// TwinCAT 3 PLC project lighting
// ProgramVersion: 3.1.4023.0
// libraries:
//   Tc2_Standard, * (Beckhoff Automation GmbH)
//   Tc2_System, * (Beckhoff Automation GmbH)
//   Tc2_Utilities, * (Beckhoff Automation GmbH)
//   Tc3_EventLogger, * (Beckhoff Automation GmbH)
//   Tc3_Module, * (Beckhoff Automation GmbH)
//   VisuDialogs, * (System)
//   Tc3_DALI,3.13.0.0,Beckhoff Automation GmbH
// project tree:
//   Bridge/ FB_DALIBridge.TcPOU, GVL_DALIBridge.TcGVL
//   Bridge/Types/ E_DALIBridgeCommand.TcTLEO, ST_DALIBridgeInputEvent.TcDUT, ST_DALIBridgeInputEventParams.TcDUT, ST_DALIBridgeNotification.TcDUT, ST_DALIBridgeRequest.TcDUT, ST_DALIBridgeResponse.TcDUT, U_ReinterpretDALIEnum.TcDUT
//   / BRIDGE_TASK.TcTTO, GlobalTextList.TcGTLO
//   GVLs/ GVL_Bridges.TcGVL, GVL_Variant.TcGVL
//   POUs/ MAIN.TcPOU
//   Tc3_DALI_PLC_Commissioning_Tool/ COMM_TASK.TcTTO, GlobalTextList_1.TcGTLO, ImagePool.TcIPO (not stored), VisualizationManager.TcVMO (not stored), VISU_TASK.TcTTO
//   Tc3_DALI_PLC_Commissioning_Tool/DUTs/ E_DALIExtendedFadeTime.TcTLEO, ST_DALI102Parameters.TcDUT, ST_DALI103Parameters.TcDUT, ST_DALIMemoryBank.TcDUT
//   Tc3_DALI_PLC_Commissioning_Tool/GVLs/ GVL.TcGVL, GVL_Internal.TcGVL
//   Tc3_DALI_PLC_Commissioning_Tool/POUs/ Communication.TcPOU, DALI_Commissioning.TcPOU, MAIN_Comissioning.TcPOU
//   Tc3_DALI_PLC_Commissioning_Tool/POUs/DALI_PLC_Commissioning/ FB_Part102Addressing.TcPOU, FB_Part102Commands.TcPOU (not stored), FB_Part102Groups.TcPOU, FB_Part102MemoryPages.TcPOU, FB_Part102Parameters.TcPOU, FB_Part102Scenes.TcPOU, FB_Part102SetFading.TcPOU, FB_Part103Addressing.TcPOU, FB_Part103MemoryPages.TcPOU, FB_Part103Parameters.TcPOU, FB_Part207ParametersLED.TcPOU, FB_Part207StatusLED.TcPOU, FB_Part300GenericDevice.TcPOU, FB_Part301PushButton.TcPOU, FB_Part302AbsoluteInputDevice.TcPOU, FB_Part303OccupancySensor.TcPOU, FB_Part304LightSensor.TcPOU
//   Tc3_DALI_PLC_Commissioning_Tool/Version/ Global_Version.TcGVL
//   Tc3_DALI_PLC_Commissioning_Tool/VISUs/TextLists/ CommandOnTerminalEvent.TcTLO, DimmingCurve.TcTLO, EventPriority.TcTLO, EventScheme.TcTLO, ExtendedFadeTime.TcTLO, FadeRate.TcTLO, FadeTime.TcTLO, FastFadeTime.TcTLO, TextList_Dialogs.TcTLO
//   Tc3_DALI_PLC_Commissioning_Tool/VISUs/ Visu_DALICommissioning.TcVIS
//   Tc3_DALI_PLC_Commissioning_Tool/VISUs/Visu_DALICommissioning/ Visu_KL6821Configuration.TcVIS, Visu_Part102Addressing.TcVIS, Visu_Part102Commands.TcVIS, Visu_Part102Groups.TcVIS, Visu_Part102MemoryBank.TcVIS, Visu_Part102Parameters.TcVIS, Visu_Part102Scenes.TcVIS, Visu_Part102SetFading.TcVIS, Visu_Part103Addressing.TcVIS, Visu_Part103MemoryBank.TcVIS, Visu_Part103Parameters.TcVIS, Visu_Part207Parameters.TcVIS, Visu_Part207Status.TcVIS, Visu_Part300GenericDevice.TcVIS, Visu_Part301PushButton.TcVIS, Visu_Part302AbsoluteInputDevice.TcVIS, Visu_Part303OccupancySensor.TcVIS, Visu_Part304LightSensor.TcVIS
// real-time tasks:
//   TASK VISU_TASK: cycle T#80ms, priority 30, ADS port 353
//   TASK BRIDGE_TASK: cycle T#8ms, priority 3, ADS port 350
//   TASK COMM_TASK: cycle T#2ms, priority 2, ADS port 351
// I/O:
//   DEVICE Device 1 (EtherCAT), AmsNetId 5.109.178.35.2.1
//     Term 1 (EK1200) [EK1200-5000 EtherCAT Power supply (2A E-Bus)]
//       Junction 1 (EK1122) [EK1122 2 port EtherCAT junction] (disabled)
//         Tenant 1 Coupler (BK1150) (disabled)
//         Tenant 2 Coupler (BK1150)
//       Junction 2  (EK1122) [EK1122 2 port EtherCAT junction] (disabled)
//         Tenant 3 Coupler (BK1150)
//         Tenant 4 Coupler (BK1150)
//       Junction 3 (EK1122) [EK1122 2 port EtherCAT junction]
//         Life Safety Coupler (BK1150) (disabled)
//       Landlord Coupler (BK1250)
// variable links:
//   lighting Instance <-> Device 1 (EtherCAT)/Term 1 (EK1200)/Junction 1 (EK1122)/Tenant 1 Coupler (BK1150)
//     COMM_TASK Inputs/GVL.aKL6821InData[1] @bit 16 <-> T1 Bus 1 (KL6821)/Channel 1/Data In 0
//     COMM_TASK Inputs/GVL.aKL6821InData[1] @bit 24 <-> T1 Bus 1 (KL6821)/Channel 1/Data In 1
//     COMM_TASK Inputs/GVL.aKL6821InData[1] @bit 32 <-> T1 Bus 1 (KL6821)/Channel 1/Data In 2
//     COMM_TASK Inputs/GVL.aKL6821InData[1] @bit 40 <-> T1 Bus 1 (KL6821)/Channel 1/Data In 3
//     COMM_TASK Inputs/GVL.aKL6821InData[2] @bit 16 <-> T1 Bus 2 (KL6821)/Channel 1/Data In 0
//     COMM_TASK Inputs/GVL.aKL6821InData[2] @bit 24 <-> T1 Bus 2 (KL6821)/Channel 1/Data In 1
//     COMM_TASK Inputs/GVL.aKL6821InData[2] @bit 32 <-> T1 Bus 2 (KL6821)/Channel 1/Data In 2
//     COMM_TASK Inputs/GVL.aKL6821InData[2] @bit 40 <-> T1 Bus 2 (KL6821)/Channel 1/Data In 3
//     COMM_TASK Inputs/GVL.aKL6821InData[1] <-> T1 Bus 1 (KL6821)/Channel 1/State
//     COMM_TASK Inputs/GVL.aKL6821InData[2] <-> T1 Bus 2 (KL6821)/Channel 1/State
//     COMM_TASK Outputs/GVL.aKL6821OutData[1] <-> T1 Bus 1 (KL6821)/Channel 1/Ctrl
//     COMM_TASK Outputs/GVL.aKL6821OutData[2] <-> T1 Bus 2 (KL6821)/Channel 1/Ctrl
//     COMM_TASK Outputs/GVL.aKL6821OutData[1] @bit 16 <-> T1 Bus 1 (KL6821)/Channel 1/Data Out 0
//     COMM_TASK Outputs/GVL.aKL6821OutData[1] @bit 24 <-> T1 Bus 1 (KL6821)/Channel 1/Data Out 1
//     COMM_TASK Outputs/GVL.aKL6821OutData[1] @bit 32 <-> T1 Bus 1 (KL6821)/Channel 1/Data Out 2
//     COMM_TASK Outputs/GVL.aKL6821OutData[1] @bit 40 <-> T1 Bus 1 (KL6821)/Channel 1/Data Out 3
//     COMM_TASK Outputs/GVL.aKL6821OutData[2] @bit 16 <-> T1 Bus 2 (KL6821)/Channel 1/Data Out 0
//     COMM_TASK Outputs/GVL.aKL6821OutData[2] @bit 24 <-> T1 Bus 2 (KL6821)/Channel 1/Data Out 1
//     COMM_TASK Outputs/GVL.aKL6821OutData[2] @bit 32 <-> T1 Bus 2 (KL6821)/Channel 1/Data Out 2
//     COMM_TASK Outputs/GVL.aKL6821OutData[2] @bit 40 <-> T1 Bus 2 (KL6821)/Channel 1/Data Out 3
//   lighting Instance <-> Device 1 (EtherCAT)/Term 1 (EK1200)/Junction 1 (EK1122)/Tenant 2 Coupler (BK1150)
//     COMM_TASK Inputs/GVL.aKL6821InData[3] @bit 16 <-> T2 Bus 1 (KL6821)/Channel 1/Data In 0
//     COMM_TASK Inputs/GVL.aKL6821InData[3] @bit 24 <-> T2 Bus 1 (KL6821)/Channel 1/Data In 1
//     COMM_TASK Inputs/GVL.aKL6821InData[3] @bit 32 <-> T2 Bus 1 (KL6821)/Channel 1/Data In 2
//     COMM_TASK Inputs/GVL.aKL6821InData[3] @bit 40 <-> T2 Bus 1 (KL6821)/Channel 1/Data In 3
//     COMM_TASK Inputs/GVL.aKL6821InData[5] @bit 16 <-> T2 Bus 3 (KL6821)/Channel 1/Data In 0
//     COMM_TASK Inputs/GVL.aKL6821InData[5] @bit 24 <-> T2 Bus 3 (KL6821)/Channel 1/Data In 1
//     COMM_TASK Inputs/GVL.aKL6821InData[5] @bit 32 <-> T2 Bus 3 (KL6821)/Channel 1/Data In 2
//     COMM_TASK Inputs/GVL.aKL6821InData[5] @bit 40 <-> T2 Bus 3 (KL6821)/Channel 1/Data In 3
//     COMM_TASK Inputs/GVL.aKL6821InData[3] <-> T2 Bus 1 (KL6821)/Channel 1/State
//     COMM_TASK Inputs/GVL.aKL6821InData[5] <-> T2 Bus 3 (KL6821)/Channel 1/State
//     COMM_TASK Inputs/GVL.aKL6821InData[4]/aData[{0..3}] <-> T2 Bus 2 (KL6821)/Channel 1/Data In {0..3}  (4 links)
//     COMM_TASK Inputs/GVL.aKL6821InData[4]/nStatus <-> T2 Bus 2 (KL6821)/Channel 1/State
//     COMM_TASK Outputs/GVL.aKL6821OutData[3] <-> T2 Bus 1 (KL6821)/Channel 1/Ctrl
//     COMM_TASK Outputs/GVL.aKL6821OutData[4] <-> T2 Bus 2 (KL6821)/Channel 1/Ctrl
//     COMM_TASK Outputs/GVL.aKL6821OutData[5] <-> T2 Bus 3 (KL6821)/Channel 1/Ctrl
//     COMM_TASK Outputs/GVL.aKL6821OutData[3] @bit 16 <-> T2 Bus 1 (KL6821)/Channel 1/Data Out 0
//     COMM_TASK Outputs/GVL.aKL6821OutData[3] @bit 24 <-> T2 Bus 1 (KL6821)/Channel 1/Data Out 1
//     COMM_TASK Outputs/GVL.aKL6821OutData[3] @bit 32 <-> T2 Bus 1 (KL6821)/Channel 1/Data Out 2
//     COMM_TASK Outputs/GVL.aKL6821OutData[3] @bit 40 <-> T2 Bus 1 (KL6821)/Channel 1/Data Out 3
//     COMM_TASK Outputs/GVL.aKL6821OutData[4] @bit 16 <-> T2 Bus 2 (KL6821)/Channel 1/Data Out 0
//     COMM_TASK Outputs/GVL.aKL6821OutData[4] @bit 24 <-> T2 Bus 2 (KL6821)/Channel 1/Data Out 1
//     COMM_TASK Outputs/GVL.aKL6821OutData[4] @bit 32 <-> T2 Bus 2 (KL6821)/Channel 1/Data Out 2
//     COMM_TASK Outputs/GVL.aKL6821OutData[4] @bit 40 <-> T2 Bus 2 (KL6821)/Channel 1/Data Out 3
//     COMM_TASK Outputs/GVL.aKL6821OutData[5] @bit 16 <-> T2 Bus 3 (KL6821)/Channel 1/Data Out 0
//     COMM_TASK Outputs/GVL.aKL6821OutData[5] @bit 24 <-> T2 Bus 3 (KL6821)/Channel 1/Data Out 1
//     COMM_TASK Outputs/GVL.aKL6821OutData[5] @bit 32 <-> T2 Bus 3 (KL6821)/Channel 1/Data Out 2
//     COMM_TASK Outputs/GVL.aKL6821OutData[5] @bit 40 <-> T2 Bus 3 (KL6821)/Channel 1/Data Out 3
//   lighting Instance <-> Device 1 (EtherCAT)/Term 1 (EK1200)/Junction 2  (EK1122)/Tenant 3 Coupler (BK1150)
//     COMM_TASK Inputs/GVL.aKL6821InData[6] @bit 16 <-> T3 Bus 1 (KL6821)/Channel 1/Data In 0
//     COMM_TASK Inputs/GVL.aKL6821InData[6] @bit 24 <-> T3 Bus 1 (KL6821)/Channel 1/Data In 1
//     COMM_TASK Inputs/GVL.aKL6821InData[6] @bit 32 <-> T3 Bus 1 (KL6821)/Channel 1/Data In 2
//     COMM_TASK Inputs/GVL.aKL6821InData[6] @bit 40 <-> T3 Bus 1 (KL6821)/Channel 1/Data In 3
//     COMM_TASK Inputs/GVL.aKL6821InData[7] @bit 16 <-> T3 Bus 2 (KL6821)/Channel 1/Data In 0
//     COMM_TASK Inputs/GVL.aKL6821InData[7] @bit 24 <-> T3 Bus 2 (KL6821)/Channel 1/Data In 1
//     COMM_TASK Inputs/GVL.aKL6821InData[7] @bit 32 <-> T3 Bus 2 (KL6821)/Channel 1/Data In 2
//     COMM_TASK Inputs/GVL.aKL6821InData[7] @bit 40 <-> T3 Bus 2 (KL6821)/Channel 1/Data In 3
//     COMM_TASK Inputs/GVL.aKL6821InData[6] <-> T3 Bus 1 (KL6821)/Channel 1/State
//     COMM_TASK Inputs/GVL.aKL6821InData[7] <-> T3 Bus 2 (KL6821)/Channel 1/State
//     COMM_TASK Outputs/GVL.aKL6821OutData[6] <-> T3 Bus 1 (KL6821)/Channel 1/Ctrl
//     COMM_TASK Outputs/GVL.aKL6821OutData[7] <-> T3 Bus 2 (KL6821)/Channel 1/Ctrl
//     COMM_TASK Outputs/GVL.aKL6821OutData[6] @bit 16 <-> T3 Bus 1 (KL6821)/Channel 1/Data Out 0
//     COMM_TASK Outputs/GVL.aKL6821OutData[6] @bit 24 <-> T3 Bus 1 (KL6821)/Channel 1/Data Out 1
//     COMM_TASK Outputs/GVL.aKL6821OutData[6] @bit 32 <-> T3 Bus 1 (KL6821)/Channel 1/Data Out 2
//     COMM_TASK Outputs/GVL.aKL6821OutData[6] @bit 40 <-> T3 Bus 1 (KL6821)/Channel 1/Data Out 3
//     COMM_TASK Outputs/GVL.aKL6821OutData[7] @bit 16 <-> T3 Bus 2 (KL6821)/Channel 1/Data Out 0
//     COMM_TASK Outputs/GVL.aKL6821OutData[7] @bit 24 <-> T3 Bus 2 (KL6821)/Channel 1/Data Out 1
//     COMM_TASK Outputs/GVL.aKL6821OutData[7] @bit 32 <-> T3 Bus 2 (KL6821)/Channel 1/Data Out 2
//     COMM_TASK Outputs/GVL.aKL6821OutData[7] @bit 40 <-> T3 Bus 2 (KL6821)/Channel 1/Data Out 3
//   lighting Instance <-> Device 1 (EtherCAT)/Term 1 (EK1200)/Junction 2  (EK1122)/Tenant 4 Coupler (BK1150)
//     COMM_TASK Inputs/GVL.aKL6821InData[8] @bit 16 <-> T4 Bus 1 (KL6821)/Channel 1/Data In 0
//     COMM_TASK Inputs/GVL.aKL6821InData[8] @bit 24 <-> T4 Bus 1 (KL6821)/Channel 1/Data In 1
//     COMM_TASK Inputs/GVL.aKL6821InData[8] @bit 32 <-> T4 Bus 1 (KL6821)/Channel 1/Data In 2
//     COMM_TASK Inputs/GVL.aKL6821InData[8] @bit 40 <-> T4 Bus 1 (KL6821)/Channel 1/Data In 3
//     COMM_TASK Inputs/GVL.aKL6821InData[9] @bit 16 <-> T4 Bus 2 (KL6821)/Channel 1/Data In 0
//     COMM_TASK Inputs/GVL.aKL6821InData[9] @bit 24 <-> T4 Bus 2 (KL6821)/Channel 1/Data In 1
//     COMM_TASK Inputs/GVL.aKL6821InData[9] @bit 32 <-> T4 Bus 2 (KL6821)/Channel 1/Data In 2
//     COMM_TASK Inputs/GVL.aKL6821InData[9] @bit 40 <-> T4 Bus 2 (KL6821)/Channel 1/Data In 3
//     COMM_TASK Inputs/GVL.aKL6821InData[8] <-> T4 Bus 1 (KL6821)/Channel 1/State
//     COMM_TASK Inputs/GVL.aKL6821InData[9] <-> T4 Bus 2 (KL6821)/Channel 1/State
//     COMM_TASK Outputs/GVL.aKL6821OutData[8] <-> T4 Bus 1 (KL6821)/Channel 1/Ctrl
//     COMM_TASK Outputs/GVL.aKL6821OutData[9] <-> T4 Bus 2 (KL6821)/Channel 1/Ctrl
//     COMM_TASK Outputs/GVL.aKL6821OutData[8] @bit 16 <-> T4 Bus 1 (KL6821)/Channel 1/Data Out 0
//     COMM_TASK Outputs/GVL.aKL6821OutData[8] @bit 24 <-> T4 Bus 1 (KL6821)/Channel 1/Data Out 1
//     COMM_TASK Outputs/GVL.aKL6821OutData[8] @bit 32 <-> T4 Bus 1 (KL6821)/Channel 1/Data Out 2
//     COMM_TASK Outputs/GVL.aKL6821OutData[8] @bit 40 <-> T4 Bus 1 (KL6821)/Channel 1/Data Out 3
//     COMM_TASK Outputs/GVL.aKL6821OutData[9] @bit 16 <-> T4 Bus 2 (KL6821)/Channel 1/Data Out 0
//     COMM_TASK Outputs/GVL.aKL6821OutData[9] @bit 24 <-> T4 Bus 2 (KL6821)/Channel 1/Data Out 1
//     COMM_TASK Outputs/GVL.aKL6821OutData[9] @bit 32 <-> T4 Bus 2 (KL6821)/Channel 1/Data Out 2
//     COMM_TASK Outputs/GVL.aKL6821OutData[9] @bit 40 <-> T4 Bus 2 (KL6821)/Channel 1/Data Out 3
//   lighting Instance <-> Device 1 (EtherCAT)/Term 1 (EK1200)/Junction 3 (EK1122)/Life Safety Coupler (BK1150)
//     COMM_TASK Inputs/GVL.aKL6821InData[10] @bit {16..40 step 8} <-> LS Bus (KL6821)/Channel 1/Data In {0..3}  (4 links)
//     COMM_TASK Inputs/GVL.aKL6821InData[10] <-> LS Bus (KL6821)/Channel 1/State
//     COMM_TASK Outputs/GVL.aKL6821OutData[10] <-> LS Bus (KL6821)/Channel 1/Ctrl
//     COMM_TASK Outputs/GVL.aKL6821OutData[10] @bit {16..40 step 8} <-> LS Bus (KL6821)/Channel 1/Data Out {0..3}  (4 links)
//   lighting Instance <-> Device 1 (EtherCAT)/Term 1 (EK1200)/Landlord Coupler (BK1250)
//     COMM_TASK Inputs/GVL.aKL6821InData[11] @bit 16 <-> LL Bus 1 (KL6821)/Channel 1/Data In 0
//     COMM_TASK Inputs/GVL.aKL6821InData[11] @bit 24 <-> LL Bus 1 (KL6821)/Channel 1/Data In 1
//     COMM_TASK Inputs/GVL.aKL6821InData[11] @bit 32 <-> LL Bus 1 (KL6821)/Channel 1/Data In 2
//     COMM_TASK Inputs/GVL.aKL6821InData[11] @bit 40 <-> LL Bus 1 (KL6821)/Channel 1/Data In 3
//     COMM_TASK Inputs/GVL.aKL6821InData[12] @bit 16 <-> LL Bus 2 (KL6821)/Channel 1/Data In 0
//     COMM_TASK Inputs/GVL.aKL6821InData[12] @bit 24 <-> LL Bus 2 (KL6821)/Channel 1/Data In 1
//     COMM_TASK Inputs/GVL.aKL6821InData[12] @bit 32 <-> LL Bus 2 (KL6821)/Channel 1/Data In 2
//     COMM_TASK Inputs/GVL.aKL6821InData[12] @bit 40 <-> LL Bus 2 (KL6821)/Channel 1/Data In 3
//     COMM_TASK Inputs/GVL.aKL6821InData[13] @bit 16 <-> LL Bus 3 (KL6821)/Channel 1/Data In 0
//     COMM_TASK Inputs/GVL.aKL6821InData[13] @bit 24 <-> LL Bus 3 (KL6821)/Channel 1/Data In 1
//     COMM_TASK Inputs/GVL.aKL6821InData[13] @bit 32 <-> LL Bus 3 (KL6821)/Channel 1/Data In 2
//     COMM_TASK Inputs/GVL.aKL6821InData[13] @bit 40 <-> LL Bus 3 (KL6821)/Channel 1/Data In 3
//     COMM_TASK Inputs/GVL.aKL6821InData[14] @bit 16 <-> LL Bus 4 (KL6821)/Channel 1/Data In 0
//     COMM_TASK Inputs/GVL.aKL6821InData[14] @bit 24 <-> LL Bus 4 (KL6821)/Channel 1/Data In 1
//     COMM_TASK Inputs/GVL.aKL6821InData[14] @bit 32 <-> LL Bus 4 (KL6821)/Channel 1/Data In 2
//     COMM_TASK Inputs/GVL.aKL6821InData[14] @bit 40 <-> LL Bus 4 (KL6821)/Channel 1/Data In 3
//     COMM_TASK Inputs/GVL.aKL6821InData[15] @bit 16 <-> LL Bus 5 (KL6821)/Channel 1/Data In 0
//     COMM_TASK Inputs/GVL.aKL6821InData[15] @bit 24 <-> LL Bus 5 (KL6821)/Channel 1/Data In 1
//     COMM_TASK Inputs/GVL.aKL6821InData[15] @bit 32 <-> LL Bus 5 (KL6821)/Channel 1/Data In 2
//     COMM_TASK Inputs/GVL.aKL6821InData[15] @bit 40 <-> LL Bus 5 (KL6821)/Channel 1/Data In 3
//     COMM_TASK Inputs/GVL.aKL6821InData[16] @bit 16 <-> LL Bus 6 (KL6821)/Channel 1/Data In 0
//     COMM_TASK Inputs/GVL.aKL6821InData[16] @bit 24 <-> LL Bus 6 (KL6821)/Channel 1/Data In 1
//     COMM_TASK Inputs/GVL.aKL6821InData[16] @bit 32 <-> LL Bus 6 (KL6821)/Channel 1/Data In 2
//     COMM_TASK Inputs/GVL.aKL6821InData[16] @bit 40 <-> LL Bus 6 (KL6821)/Channel 1/Data In 3
//     COMM_TASK Inputs/GVL.aKL6821InData[{11..16}] <-> LL Bus {1..6} (KL6821)/Channel 1/State  (6 links)
//     COMM_TASK Outputs/GVL.aKL6821OutData[{11..16}] <-> LL Bus {1..6} (KL6821)/Channel 1/Ctrl  (6 links)
//     COMM_TASK Outputs/GVL.aKL6821OutData[11] @bit 16 <-> LL Bus 1 (KL6821)/Channel 1/Data Out 0
//     COMM_TASK Outputs/GVL.aKL6821OutData[11] @bit 24 <-> LL Bus 1 (KL6821)/Channel 1/Data Out 1
//     COMM_TASK Outputs/GVL.aKL6821OutData[11] @bit 32 <-> LL Bus 1 (KL6821)/Channel 1/Data Out 2
//     COMM_TASK Outputs/GVL.aKL6821OutData[11] @bit 40 <-> LL Bus 1 (KL6821)/Channel 1/Data Out 3
//     COMM_TASK Outputs/GVL.aKL6821OutData[12] @bit 16 <-> LL Bus 2 (KL6821)/Channel 1/Data Out 0
//     COMM_TASK Outputs/GVL.aKL6821OutData[12] @bit 24 <-> LL Bus 2 (KL6821)/Channel 1/Data Out 1
//     COMM_TASK Outputs/GVL.aKL6821OutData[12] @bit 32 <-> LL Bus 2 (KL6821)/Channel 1/Data Out 2
//     COMM_TASK Outputs/GVL.aKL6821OutData[12] @bit 40 <-> LL Bus 2 (KL6821)/Channel 1/Data Out 3
//     COMM_TASK Outputs/GVL.aKL6821OutData[13] @bit 16 <-> LL Bus 3 (KL6821)/Channel 1/Data Out 0
//     COMM_TASK Outputs/GVL.aKL6821OutData[13] @bit 24 <-> LL Bus 3 (KL6821)/Channel 1/Data Out 1
//     COMM_TASK Outputs/GVL.aKL6821OutData[13] @bit 32 <-> LL Bus 3 (KL6821)/Channel 1/Data Out 2
//     COMM_TASK Outputs/GVL.aKL6821OutData[13] @bit 40 <-> LL Bus 3 (KL6821)/Channel 1/Data Out 3
//     COMM_TASK Outputs/GVL.aKL6821OutData[14] @bit 16 <-> LL Bus 4 (KL6821)/Channel 1/Data Out 0
//     COMM_TASK Outputs/GVL.aKL6821OutData[14] @bit 24 <-> LL Bus 4 (KL6821)/Channel 1/Data Out 1
//     COMM_TASK Outputs/GVL.aKL6821OutData[14] @bit 32 <-> LL Bus 4 (KL6821)/Channel 1/Data Out 2
//     COMM_TASK Outputs/GVL.aKL6821OutData[14] @bit 40 <-> LL Bus 4 (KL6821)/Channel 1/Data Out 3
//     COMM_TASK Outputs/GVL.aKL6821OutData[15] @bit 16 <-> LL Bus 5 (KL6821)/Channel 1/Data Out 0
//     COMM_TASK Outputs/GVL.aKL6821OutData[15] @bit 24 <-> LL Bus 5 (KL6821)/Channel 1/Data Out 1
//     COMM_TASK Outputs/GVL.aKL6821OutData[15] @bit 32 <-> LL Bus 5 (KL6821)/Channel 1/Data Out 2
//     COMM_TASK Outputs/GVL.aKL6821OutData[15] @bit 40 <-> LL Bus 5 (KL6821)/Channel 1/Data Out 3
//     COMM_TASK Outputs/GVL.aKL6821OutData[16] @bit 16 <-> LL Bus 6 (KL6821)/Channel 1/Data Out 0
//     COMM_TASK Outputs/GVL.aKL6821OutData[16] @bit 24 <-> LL Bus 6 (KL6821)/Channel 1/Data Out 1
//     COMM_TASK Outputs/GVL.aKL6821OutData[16] @bit 32 <-> LL Bus 6 (KL6821)/Channel 1/Data Out 2
//     COMM_TASK Outputs/GVL.aKL6821OutData[16] @bit 40 <-> LL Bus 6 (KL6821)/Channel 1/Data Out 3

CONFIGURATION lighting
    RESOURCE PLC ON TwinCAT3
        TASK BRIDGE_TASK(INTERVAL := T#8ms, PRIORITY := 3);
        TASK COMM_TASK(INTERVAL := T#2ms, PRIORITY := 2);
        TASK VISU_TASK(INTERVAL := T#80ms, PRIORITY := 30);
        PROGRAM MAIN WITH BRIDGE_TASK : MAIN;
        PROGRAM MAIN_Comissioning WITH BRIDGE_TASK : MAIN_Comissioning;
        PROGRAM Communication WITH COMM_TASK : Communication;
        PROGRAM VisuElems_Visu_Prg WITH VISU_TASK : VisuElems.Visu_Prg;
    END_RESOURCE
END_CONFIGURATION

// ---- Bridge/Types/E_DALIBridgeCommand.TcTLEO
{attribute 'qualified_only'}
{attribute 'strict'}
TYPE E_DALIBridgeCommand :
(
	idle						:= 0,
	directArcPowerControl		:= 1,
	queryActualLevel			:= 2,
	queryStatus					:= 3,
	setEventScheme				:= 4,
	queryEventScheme			:= 5,
	setEventFilter				:= 6,
	queryEventFilter			:= 7,
	identifyDevice102			:= 8,
	identifyDevice103			:= 9,
	enableInstance				:= 10,
	goToScene					:= 11,
	setFadeTime					:= 12,
	queryInputValue				:= 13,
	queryBatteryCharge			:= 14,
	queryDurationTestResult		:= 15,
	queryEmergencyMode			:= 16,
	queryEmergencyStatus		:= 17,
	queryFailureStatus			:= 18,
	queryRatedDuration			:= 19,
	queryTestTiming				:= 20,
	resetDurationTestDoneFlag	:= 21,
	resetFunctionTestDoneFlag	:= 22,
	startDurationTest			:= 23,
	startFunctionTest			:= 24,
	stopTest					:= 25,
	setDurationTestInterval		:= 26,
	setFunctionTestInterval		:= 27,
	startIdentification202		:= 28,
	queryGroups					:= 29,
	addToGroup					:= 30,
	removeFromGroup				:= 31,
	enabledDeviceType			:= 32,
	
	testCommand := 100
);
END_TYPE

// ---- Bridge/Types/ST_DALIBridgeInputEvent.TcDUT
TYPE ST_DALIBridgeInputEvent :
STRUCT
	parameters : ST_DALIBridgeInputEventParams;
	error      : BOOL;
	status     : UDINT;
	message    : STRING(255);
	data       : WORD;
END_STRUCT
END_TYPE

// ---- Bridge/Types/ST_DALIBridgeInputEventParams.TcDUT
TYPE ST_DALIBridgeInputEventParams :
STRUCT
	eventScheme 	: E_DALIEventScheme;
	addressInfo1 	: BYTE;
	addressInfo2 	: BYTE;
END_STRUCT
END_TYPE

// ---- Bridge/Types/ST_DALIBridgeNotification.TcDUT
TYPE ST_DALIBridgeNotification :
STRUCT
	valid 				: BOOL;
	sequence 			: ULINT;
	nInputEvents		: BYTE;
	inputEvents 		: ARRAY [0..GVL_DALIBridge.maxInputEventsPerNotification-1] OF ST_DALIBridgeInputEvent;
END_STRUCT
END_TYPE

// ---- Bridge/Types/ST_DALIBridgeRequest.TcDUT
TYPE ST_DALIBridgeRequest :
STRUCT
	command 			: E_DALIBridgeCommand := E_DALIBridgeCommand.idle;
	address 			: BYTE;
	addressType 		: E_DALIAddressType;
	instanceAddress 	: BYTE;
	instanceAddressType : E_DALIInstanceAddressType;
	data            	: BYTE;
END_STRUCT
END_TYPE

// ---- Bridge/Types/ST_DALIBridgeResponse.TcDUT
TYPE ST_DALIBridgeResponse :
STRUCT
	valid       : BOOL := FALSE; 	// True if the struct contains valid data.
	sequence 	: ULINT;			// Same as the sequence number returned when calling RpcRequest
	error       : BOOL;				// True if an error condition ocurred. If error is false but status is nonzero, a warning occurred.
	status      : UDINT;			// Status code returned by the operation
	message     : STRING(255);		// Human-readable error message
	data 		: LWORD;			// Data returned by a DALI read command. If the command does not read data, then ignore this field.
END_STRUCT
END_TYPE

// ---- Bridge/Types/U_ReinterpretDALIEnum.TcDUT
TYPE U_ReinterpretDALIEnum :
UNION
	raw				: BYTE;
	eventScheme 	: E_DALIEventScheme;
	fadeTime		: E_DALIFadeTime;
	testTiming      : E_DALITestTiming;
	deviceType		: E_DALIDeviceType;
END_UNION
END_TYPE

// ---- Tc3_DALI_PLC_Commissioning_Tool/DUTs/E_DALIExtendedFadeTime.TcTLEO
{attribute 'qualified_only'}
{attribute 'strict'}
TYPE E_DALIExtendedFadeTime :
(
	NoFade := 0,
	onehundred := 1,
	twohundred := 2,
	threehundred := 3,
	fourhundred := 4,
	fivehundred := 5,
	sixhundred := 6,
	sevenhundred := 7,
	eighthundred := 8,
	ninehundred := 9,
	onethousand := 10,
	onethousandonehundred := 11,
	onethousandtwohundred := 12,
	onethousandthreehundred := 13,
	onethousandfourhundred := 14,
	onethousandfivehundred := 15,
	onethousandsixhundred	:= 16,
	onesecond := 17,
	twoseconds := 18,
	threeseconds := 19,
	fourseconds := 20,
	fiveseconds := 21,
	sixseconds := 22,
	sevenseconds := 23,
	eightseconds := 24,
	nineseconds := 25,
	tenseconds := 26,
	elevenseconds := 27,
	twelveseconds := 28,
	thirteenseconds := 29,
	fourteenseconds := 30,
	fifteenseconds := 31,
	sixteenseconds := 32,
	ten1seconds := 33,
	twentyseconds := 34,
	thirtyseconds := 35,
	fourtyseconds := 36,
	fiftyseconds := 37,
	sixtyseconds := 38,
	seventyseconds := 39,
	eightyseconds := 40,
	ninetyseconds := 41,
	onehundredseconds := 42,
	onehundredtenseconds := 43,
	onehundredtwentyseconds := 44,
	onehundredthirtyseconds := 45,
	onehundredfourtyseconds := 46,
	onehundredfiftyseconds := 47,
	onehundredsixtyseconds := 48,
	oneminute := 49,
	twominutes := 50,
	threeminutes := 51,
	fourminutes := 52,
	fiveminutes := 53,
	sixminutes := 54,
	sevenminutes := 55,
	eightminutes := 56,
	nineminutes := 57,
	tenminutes := 58,
	elevenminutes := 59,
	twelveminutes := 60,
	thirteenminutes := 61,
	fourteenminutes := 62,
	fifteenminutes := 63,
	sixteenminutes := 64,
	unknown := 255
);
END_TYPE

// ---- Tc3_DALI_PLC_Commissioning_Tool/DUTs/ST_DALI102Parameters.TcDUT
TYPE ST_DALI102Parameters :
STRUCT
	nShortAddress			:	BYTE; // 255: no short address
	nActualLevel			:	BYTE;
	nMinLevel				:	BYTE;
	nMaxLevel				: 	BYTE;
	eFadeRate				:	E_DALIFadeRate;
	eFadeTime				:	E_DALIFadeTime;
	nPowerOnLevel			:	BYTE;
	nSystemFailureLevel		:	BYTE;
	nPhysicalMinimum		:	BYTE;
	sDeviceTypes			:	STRING[100];
END_STRUCT
END_TYPE

// ---- Tc3_DALI_PLC_Commissioning_Tool/DUTs/ST_DALI103Parameters.TcDUT
TYPE ST_DALI103Parameters :
STRUCT
	nOperatingMode			:	BYTE;
	sInstanceType0			:	STRING;
	sInstanceType1			:	STRING;
	sInstanceType2			:	STRING;
	sInstanceType3			:	STRING;
	sInstanceType4			:	STRING;
END_STRUCT
END_TYPE

// ---- Tc3_DALI_PLC_Commissioning_Tool/DUTs/ST_DALIMemoryBank.TcDUT
TYPE ST_DALIMemoryBank :
STRUCT
	sOffset			:	STRING(20);
	sName			:	STRING(255);
	nValueDec		:	BYTE;
	nValueHex		:	STRING(20);
END_STRUCT
END_TYPE

// ---- Bridge/GVL_DALIBridge.TcGVL
{attribute 'qualified_only'}
VAR_GLOBAL

END_VAR
VAR_GLOBAL CONSTANT
	maxInputEventListeners: INT := 64;
	maxInputEventsPerNotification: INT := 4;
END_VAR

// ---- GVLs/GVL_Bridges.TcGVL
{attribute 'qualified_only'}
VAR_GLOBAL
	// Landlord Buses
	bus_LL1_bridge			: FB_DALIBridge(Communication.aKL6821Communication[11]);
	bus_LL1_response		: ST_DALIBridgeResponse;
	bus_LL1_notification	: ST_DALIBridgeNotification;
	
	bus_LL2_bridge			: FB_DALIBridge(Communication.aKL6821Communication[12]);
	bus_LL2_response		: ST_DALIBridgeResponse;
	bus_LL2_notification	: ST_DALIBridgeNotification;
	
	bus_LL3_bridge			: FB_DALIBridge(Communication.aKL6821Communication[13]);
	bus_LL3_response		: ST_DALIBridgeResponse;
	bus_LL3_notification	: ST_DALIBridgeNotification;
	
	bus_LL4_bridge			: FB_DALIBridge(Communication.aKL6821Communication[14]);
	bus_LL4_response		: ST_DALIBridgeResponse;
	bus_LL4_notification	: ST_DALIBridgeNotification;
	
	bus_LL5_bridge			: FB_DALIBridge(Communication.aKL6821Communication[15]);
	bus_LL5_response		: ST_DALIBridgeResponse;
	bus_LL5_notification	: ST_DALIBridgeNotification;
	
	bus_LL6_bridge			: FB_DALIBridge(Communication.aKL6821Communication[16]);
	bus_LL6_response		: ST_DALIBridgeResponse;
	bus_LL6_notification	: ST_DALIBridgeNotification;
	
	// Life Safety Riser Bus
	bus_LS_bridge			: FB_DALIBridge(Communication.aKL6821Communication[10]);
	bus_LS_response			: ST_DALIBridgeResponse;
	bus_LS_notification		: ST_DALIBridgeNotification;
	
	// Tenant 1 Buses
	bus_T1_1_bridge			: FB_DALIBridge(Communication.aKL6821Communication[1]);
	bus_T1_1_response		: ST_DALIBridgeResponse;
	bus_T1_1_notification	: ST_DALIBridgeNotification;
	
	bus_T1_2_bridge			: FB_DALIBridge(Communication.aKL6821Communication[2]);
	bus_T1_2_response		: ST_DALIBridgeResponse;
	bus_T1_2_notification	: ST_DALIBridgeNotification;
	
	// Tenant 2 Buses
	bus_T2_1_bridge			: FB_DALIBridge(Communication.aKL6821Communication[3]);
	bus_T2_1_response		: ST_DALIBridgeResponse;
	bus_T2_1_notification	: ST_DALIBridgeNotification;
	
	bus_T2_2_bridge			: FB_DALIBridge(Communication.aKL6821Communication[4]);
	bus_T2_2_response		: ST_DALIBridgeResponse;
	bus_T2_2_notification	: ST_DALIBridgeNotification;
	
	bus_T2_3_bridge			: FB_DALIBridge(Communication.aKL6821Communication[5]);
	bus_T2_3_response		: ST_DALIBridgeResponse;
	bus_T2_3_notification	: ST_DALIBridgeNotification;
	
	// Tenant 3 Buses
	bus_T3_1_bridge			: FB_DALIBridge(Communication.aKL6821Communication[6]);
	bus_T3_1_response		: ST_DALIBridgeResponse;
	bus_T3_1_notification	: ST_DALIBridgeNotification;
	
	bus_T3_2_bridge			: FB_DALIBridge(Communication.aKL6821Communication[7]);
	bus_T3_2_response		: ST_DALIBridgeResponse;
	bus_T3_2_notification	: ST_DALIBridgeNotification;
	
	// Tenant 4 Buses
	bus_T4_1_bridge			: FB_DALIBridge(Communication.aKL6821Communication[8]);
	bus_T4_1_response		: ST_DALIBridgeResponse;
	bus_T4_1_notification	: ST_DALIBridgeNotification;
	
	bus_T4_2_bridge			: FB_DALIBridge(Communication.aKL6821Communication[9]);
	bus_T4_2_response		: ST_DALIBridgeResponse;
	bus_T4_2_notification	: ST_DALIBridgeNotification;
END_VAR

// ---- GVLs/GVL_Variant.TcGVL
{attribute 'qualified_only'}
VAR_GLOBAL CONSTANT
	{IF defined(Floor_00)}
		numLLBus 	: INT := 6;
		numT1Bus	: INT := 2;
		numT2Bus	: INT := 3;
		numT3Bus	: INT := 0;
		numT4Bus	: INT := 4;
		hasLSBus	: BOOL := FALSE;
	{ELSIF defined(Floor_01)}
		numLLBus 	: INT := 0;
		numT1Bus	: INT := 2;
		numT2Bus	: INT := 2;
		numT3Bus	: INT := 2;
		numT4Bus	: INT := 1;
		hasLSBus	: BOOL := TRUE;
	{ELSIF defined(Floor_02)}
		numLLBus 	: INT := 3;
		numT1Bus	: INT := 2;
		numT2Bus	: INT := 2;
		numT3Bus	: INT := 2;
		numT4Bus	: INT := 2;
		hasLSBus	: BOOL := FALSE;
	{ELSIF defined(Floor_03)}
		numLLBus 	: INT := 0;
		numT1Bus	: INT := 2;
		numT2Bus	: INT := 2;
		numT3Bus	: INT := 2;
		numT4Bus	: INT := 2;
		hasLSBus	: BOOL := FALSE;
	{ELSIF defined(Floor_04)}
		numLLBus 	: INT := 3;
		numT1Bus	: INT := 2;
		numT2Bus	: INT := 2;
		numT3Bus	: INT := 2;
		numT4Bus	: INT := 2;
		hasLSBus	: BOOL := TRUE;
	{ELSIF defined(Floor_05)}
		numLLBus 	: INT := 0;
		numT1Bus	: INT := 2;
		numT2Bus	: INT := 2;
		numT3Bus	: INT := 2;
		numT4Bus	: INT := 2;
		hasLSBus	: BOOL := FALSE;
	{ELSIF defined(Floor_06)}
		numLLBus 	: INT := 2;
		numT1Bus	: INT := 2;
		numT2Bus	: INT := 2;
		numT3Bus	: INT := 2;
		numT4Bus	: INT := 2;
		hasLSBus	: BOOL := FALSE;
	{ELSIF defined(Floor_07)}
		numLLBus 	: INT := 0;
		numT1Bus	: INT := 2;
		numT2Bus	: INT := 2;
		numT3Bus	: INT := 2;
		numT4Bus	: INT := 2;
		hasLSBus	: BOOL := TRUE;
	{ELSIF defined(Floor_08)}
		numLLBus 	: INT := 3;
		numT1Bus	: INT := 2;
		numT2Bus	: INT := 2;
		numT3Bus	: INT := 2;
		numT4Bus	: INT := 1;
		hasLSBus	: BOOL := FALSE;
	{ELSIF defined(Floor_09)}
		numLLBus 	: INT := 0;
		numT1Bus	: INT := 2;
		numT2Bus	: INT := 2;
		numT3Bus	: INT := 2;
		numT4Bus	: INT := 1;
		hasLSBus	: BOOL := FALSE;
	{ELSIF defined(Floor_10)}
		numLLBus 	: INT := 4;
		numT1Bus	: INT := 0;
		numT2Bus	: INT := 0;
		numT3Bus	: INT := 0;
		numT4Bus	: INT := 0;
		hasLSBus	: BOOL := FALSE;
	{ELSIF defined(Lab)}
		numLLBus 	: INT := 6;
		numT1Bus	: INT := 0;
		numT2Bus	: INT := 0;
		numT3Bus	: INT := 0;
		numT4Bus	: INT := 0;
		hasLSBus	: BOOL := TRUE;
	{ELSE}
		numLLBus 	: INT := 0;
		numT1Bus	: INT := 0;
		numT2Bus	: INT := 0;
		numT3Bus	: INT := 0;
		numT4Bus	: INT := 0;
		hasLSBus	: BOOL := FALSE;
	{END_IF}
END_VAR

// ---- Tc3_DALI_PLC_Commissioning_Tool/GVLs/GVL.TcGVL
{attribute 'qualified_only'}
VAR_GLOBAL
	{attribute 'TcContextName' := 'PlcCommunication'}
	aKL6821InData			AT %I* 	: ARRAY [1..GVL_Internal.nNumberOfDALI_Lines] OF Tc3_DALI.ST_KL6821InData;
	{attribute 'TcContextName' := 'PlcCommunication'}
	aKL6821OutData			AT %Q* 	: ARRAY [1..GVL_Internal.nNumberOfDALI_Lines] OF Tc3_DALI.ST_KL6821OutData;
END_VAR

// ---- Tc3_DALI_PLC_Commissioning_Tool/GVLs/GVL_Internal.TcGVL
{attribute 'qualified_only'}
VAR_GLOBAL
	nDALILine				:	INT := 1; // Start with DALI-Line 1 as default.
END_VAR
VAR_GLOBAL CONSTANT
	nNumberOfDALI_Lines		: 	INT := 16; // Constant to vary with the number of required DALI Lines.
END_VAR

// ---- Tc3_DALI_PLC_Commissioning_Tool/Version/Global_Version.TcGVL
{attribute 'TcGenerated'}
{attribute 'no-analysis'}
{attribute 'linkalways'}
// This function has been automatically generated from the project information.
VAR_GLOBAL CONSTANT
	{attribute 'const_non_replaced'}
	stLibVersion_Tc3_DALI_PLC_Commissioning_Tool : ST_LibVersion := (iMajor := 3, iMinor := 7, iBuild := 1, iRevision := 0, nFlags := 0, sVersion := '3.7.1.0');
END_VAR

// ---- POUs/MAIN.TcPOU
PROGRAM MAIN
VAR
	emergency : BOOL := FALSE;
END_VAR

Tc3_DALI.GVL.eEventTraceLevel := TcEventSeverity.Verbose;

// Landlord buses
IF (GVL_Variant.numLLBus >= 1) THEN
    GVL_Bridges.bus_LL1_bridge(
        emergency:= emergency,
        rpcResponse     => GVL_Bridges.bus_LL1_response,
        notification=> GVL_Bridges.bus_LL1_notification
    );
END_IF
IF (GVL_Variant.numLLBus >= 2) THEN
    GVL_Bridges.bus_LL2_bridge(
        emergency:= emergency,
        rpcResponse     => GVL_Bridges.bus_LL2_response,
        notification=> GVL_Bridges.bus_LL2_notification
    );
END_IF
IF (GVL_Variant.numLLBus >= 3) THEN
    GVL_Bridges.bus_LL3_bridge(
        emergency:= emergency,
        rpcResponse     => GVL_Bridges.bus_LL3_response,
        notification=> GVL_Bridges.bus_LL3_notification
    );
END_IF
IF (GVL_Variant.numLLBus >= 4) THEN
    GVL_Bridges.bus_LL4_bridge(
        emergency:= emergency,
        rpcResponse     => GVL_Bridges.bus_LL4_response,
        notification=> GVL_Bridges.bus_LL4_notification
    );
END_IF
IF (GVL_Variant.numLLBus >= 5) THEN
    GVL_Bridges.bus_LL5_bridge(
        emergency:= emergency,
        rpcResponse     => GVL_Bridges.bus_LL5_response,
        notification=> GVL_Bridges.bus_LL5_notification
    );
END_IF
IF (GVL_Variant.numLLBus >= 6) THEN
    GVL_Bridges.bus_LL6_bridge(
        emergency:= emergency,
        rpcResponse     => GVL_Bridges.bus_LL6_response,
        notification=> GVL_Bridges.bus_LL6_notification
    );
END_IF

// Tenant 1
IF (GVL_Variant.numT1Bus >= 1) THEN
        GVL_Bridges.bus_T1_1_bridge(
                emergency:= emergency,
                rpcResponse=> GVL_Bridges.bus_T1_1_response,
                notification=> GVL_Bridges.bus_T1_1_notification
        );
END_IF
IF (GVL_Variant.numT1Bus >= 2) THEN
        GVL_Bridges.bus_T1_2_bridge(
                emergency:= emergency,
                rpcResponse=> GVL_Bridges.bus_T1_2_response,
                notification=> GVL_Bridges.bus_T1_2_notification
        );
END_IF

// Tenant 2
IF (GVL_Variant.numT2Bus >= 1) THEN
        GVL_Bridges.bus_T2_1_bridge(
                emergency:= emergency,
                rpcResponse=> GVL_Bridges.bus_T2_1_response,
                notification=> GVL_Bridges.bus_T2_1_notification
        );
END_IF
IF (GVL_Variant.numT2Bus >= 2) THEN
        GVL_Bridges.bus_T2_2_bridge(
                emergency:= emergency,
                rpcResponse=> GVL_Bridges.bus_T2_2_response,
                notification=> GVL_Bridges.bus_T2_2_notification
        );
END_IF
IF (GVL_Variant.numT2Bus >= 3) THEN
        GVL_Bridges.bus_T2_3_bridge(
                emergency:= emergency,
                rpcResponse=> GVL_Bridges.bus_T2_3_response,
                notification=> GVL_Bridges.bus_T2_3_notification
        );
END_IF

// Tenant 3
IF (GVL_Variant.numT3Bus >= 1) THEN
        GVL_Bridges.bus_T3_1_bridge(
                emergency:= emergency,
                rpcResponse=> GVL_Bridges.bus_T3_1_response,
                notification=> GVL_Bridges.bus_T3_1_notification
        );
END_IF
IF (GVL_Variant.numT3Bus >= 2) THEN
        GVL_Bridges.bus_T3_2_bridge(
                emergency:= emergency,
                rpcResponse=> GVL_Bridges.bus_T3_2_response,
                notification=> GVL_Bridges.bus_T3_2_notification
        );
END_IF

// Tenant 4
IF (GVL_Variant.numT4Bus >= 1) THEN
        GVL_Bridges.bus_T4_1_bridge(
                emergency:= emergency,
                rpcResponse=> GVL_Bridges.bus_T4_1_response,
                notification=> GVL_Bridges.bus_T4_1_notification
        );
END_IF
IF (GVL_Variant.numT4Bus >= 2) THEN
        GVL_Bridges.bus_T4_2_bridge(
                emergency:= emergency,
                rpcResponse=> GVL_Bridges.bus_T4_2_response,
                notification=> GVL_Bridges.bus_T4_2_notification
        );
END_IF

// Life Safety Riser
IF (GVL_Variant.hasLSBus) THEN
	GVL_Bridges.bus_LS_bridge(
		emergency		:= emergency,
		rpcResponse		=> GVL_Bridges.bus_LS_response,
		notification	=> GVL_Bridges.bus_LS_notification
	);
END_IF

END_PROGRAM

// ---- Tc3_DALI_PLC_Commissioning_Tool/POUs/MAIN_Comissioning.TcPOU
PROGRAM MAIN_Comissioning
VAR
END_VAR

Tc3_DALI.GVL.eEventTraceLevel := TcEventSeverity.Verbose;
DALI_Commissioning();

END_PROGRAM

// ---- Tc3_DALI_PLC_Commissioning_Tool/POUs/DALI_Commissioning.TcPOU
PROGRAM DALI_Commissioning
VAR
	{region "Visu"}
	nSelectedDialog				:	INT;
	bDisableComboBox			:	BOOL;
	{endregion}

	fbPart102Addressing			:	FB_Part102Addressing := (ipDALICommunication := Communication.aKL6821Communication[1]);
	fbPart102Commands			:	FB_Part102Commands := (ipDALICommunication := Communication.aKL6821Communication[1]);
	fbPart102Groups				:	FB_Part102Groups := (ipDALICommunication := Communication.aKL6821Communication[1]);
	fbPart102Parameters			:	FB_Part102Parameters := (ipDALICommunication :=Communication.aKL6821Communication[1]);
	fbPart102Scenes				:	FB_Part102Scenes := (ipDALICommunication := Communication.aKL6821Communication[1]);
	fbPart103Addressing			:	FB_Part103Addressing := (ipDALICommunication := Communication.aKL6821Communication[1]);
	fbPart103Parameters			:	FB_Part103Parameters := (ipDALICommunication := Communication.aKL6821Communication[1]);
	fbPart300GenericDevice		:	FB_Part300GenericDevice := (ipDALICommunication := Communication.aKL6821Communication[1]);
	fbPart301PushButton			:	FB_Part301PushButton := (ipDALICommunication := Communication.aKL6821Communication[1]);
	fbPart302AbsoluteInputDevice:	FB_Part302AbsoluteInputDevice := (ipDALICommunication := Communication.aKL6821Communication[1]);
	fbPart303OccupancySensor	:	FB_Part303OccupancySensor := (ipDALICommunication := Communication.aKL6821Communication[1]);
	fbPart304LightSensor		:	FB_Part304LightSensor := (ipDALICommunication := Communication.aKL6821Communication[1]);
	fbPart207ParametersLED		:	FB_Part207ParametersLED := (ipDALICommunication := Communication.aKL6821Communication[1]);
	fbPart207StatusLED			:	FB_Part207StatusLED := (ipDALICommunication := Communication.aKL6821Communication[1]);
	fbPart102MemoryPages		:	FB_Part102MemoryPages := (ipDALICommunication := Communication.aKL6821Communication[1]);
	fbPart103MemoryPages		:	FB_Part103MemoryPages := (ipDALICommunication :=Communication.aKL6821Communication[1]);
	fbPart102SetFading			:	FB_Part102SetFading := (ipDALICommunication := Communication.aKL6821Communication[1]);
END_VAR

CASE nSelectedDialog OF
0:
	fbPart102Commands(ipDALICommunication := Communication.aKL6821Communication[GVL_Internal.nDALILine]);

1:
	fbPart102Parameters(ipDALICommunication := Communication.aKL6821Communication[GVL_Internal.nDALILine], bBusy=> bDisableComboBox);

2:
	fbPart102Addressing(ipDALICommunication := Communication.aKL6821Communication[GVL_Internal.nDALILine], bBusy=> bDisableComboBox);

3:
	fbPart102Groups(ipDALICommunication := Communication.aKL6821Communication[GVL_Internal.nDALILine], bBusy=> bDisableComboBox);

4:
	fbPart102Scenes(ipDALICommunication := Communication.aKL6821Communication[GVL_Internal.nDALILine], bBusy=> bDisableComboBox);

5:
	fbPart102MemoryPages(ipDALICommunication := Communication.aKL6821Communication[GVL_Internal.nDALILine], bBusy=> bDisableComboBox);

6:
	fbPart102SetFading(ipDALICommunication := Communication.aKL6821Communication[GVL_Internal.nDALILine], bBusy=> bDisableComboBox);

7:
	fbPart207StatusLED(ipDALICommunication := Communication.aKL6821Communication[GVL_Internal.nDALILine], bBusy=> bDisableComboBox);

8:
	fbPart103Parameters(ipDALICommunication := Communication.aKL6821Communication[GVL_Internal.nDALILine], bBusy=> bDisableComboBox);

9:
	fbPart103Addressing(ipDALICommunication := Communication.aKL6821Communication[GVL_Internal.nDALILine], bBusy=> bDisableComboBox);

10:
	fbPart301PushButton(ipDALICommunication := Communication.aKL6821Communication[GVL_Internal.nDALILine], bBusy=> bDisableComboBox);

11:
	fbPart302AbsoluteInputDevice(ipDALICommunication := Communication.aKL6821Communication[GVL_Internal.nDALILine], bBusy=> bDisableComboBox);

12:
	fbPart303OccupancySensor(ipDALICommunication := Communication.aKL6821Communication[GVL_Internal.nDALILine], bBusy=> bDisableComboBox);

13:
	fbPart304LightSensor(ipDALICommunication := Communication.aKL6821Communication[GVL_Internal.nDALILine], bBusy=> bDisableComboBox);

14:
	fbPart300GenericDevice(ipDALICommunication := Communication.aKL6821Communication[GVL_Internal.nDALILine], bBusy=> bDisableComboBox);  

15:
	fbPart103MemoryPages(ipDALICommunication := Communication.aKL6821Communication[GVL_Internal.nDALILine], bBusy=> bDisableComboBox);

16:
	Communication.aKL6821Communication[GVL_Internal.nDALILine](stInData := GVL.aKL6821InData[GVL_Internal.nDALILine], stOutData := GVL.aKL6821OutData[GVL_Internal.nDALILine], bBusy=> bDisableComboBox);
END_CASE
{endregion}

END_PROGRAM

// ---- Tc3_DALI_PLC_Commissioning_Tool/POUs/DALI_PLC_Commissioning/FB_Part102Addressing.TcPOU
FUNCTION_BLOCK FB_Part102Addressing
VAR_INPUT
	ipDALICommunication			:	I_DALICommunication;
END_VAR
VAR_OUTPUT
	bBusy						:	BOOL;
END_VAR
VAR
	{region "Visu"}
	bScanDevices				:	BOOL;
	bStartChangeAddress			:	BOOL;
	bStartRandomAddressing		:	BOOL;
	nStartAddress				:	BYTE;
	bNewInstallation			:	BOOL;
	bOpticalFeedback			:	BOOL;
	bHideWaitSymbol				:	BOOL := TRUE;
	{endregion}
	nStep						:	INT;
	nAddress					:	INT;
	aChangeAddressList			:	ARRAY [0..63] OF ST_DALIChangeAddressList;
	aShortAddress				:	ARRAY [0..63] OF INT;
	aNoShortAddress				:	ARRAY [0..63] OF BOOL;
	nRow						:	INT;
	nHideLine					:	INT; // Variable to find out how many rows are used

	fb102Addressing				:	FB_DALI102Addressing(0);
	fb102QueryRandomAddress		:	FB_DALI102QueryRandomAddress(0);
	fb102ChangeAddresses		:	FB_DALI102ChangeAddresses(0);
END_VAR

{region "Detect Commands"}
IF (bStartRandomAddressing AND (nStep = 0)) THEN
	nStep := 10;
	bStartRandomAddressing := FALSE;
	bHideWaitSymbol := FALSE;
END_IF

IF (bScanDevices AND (nStep = 0)) THEN
	nStep := 20;
	nAddress := 0;
	bScanDevices := FALSE;
	bHideWaitSymbol := FALSE;
END_IF
	 
IF (bStartChangeAddress AND (nStep = 0)) THEN
	nStep := 60;
	bStartChangeAddress := FALSE;
	bHideWaitSymbol := FALSE;
END_IF
{endregion}
{region "Manage Dialog Selection}
IF (nStep = 0) THEN
	bBusy := FALSE;
ELSE
	bBusy := TRUE;
END_IF
{endregion}	 
{region "Execute Commands"}
CASE nStep OF
0:
{region "Init"}
	bScanDevices := FALSE;
	bStartChangeAddress := FALSE;
	bStartRandomAddressing := FALSE;
	bHideWaitSymbol := TRUE;

	fb102Addressing.ipDALICommunication := ipDALICommunication;
	fb102QueryRandomAddress.ipDALICommunication := ipDALICommunication;
	fb102ChangeAddresses.ipDALICommunication := ipDALICommunication;
{endregion}

10:
{region "Random Addressing"}
	fb102Addressing.nOptions := 0;
	
	IF bNewInstallation THEN 
		fb102Addressing.nOptions := fb102Addressing.nOptions OR Tc3_DALI.GVL.cCompleteNewInstallation;
	END_IF

	IF bOpticalFeedback THEN
		fb102Addressing.nOptions := fb102Addressing.nOptions OR Tc3_DALI.GVL.cOpticalFeedback;
	END_IF

	fb102Addressing(bStart := TRUE,
					nStartWithShortAddress := nStartAddress);
	IF (NOT fb102Addressing.bBusy) THEN
		fb102Addressing(bStart := FALSE);
		nStep := 0;
	END_IF
{endregion}
20:
{region "Read Existing Addresses"}
	// Query of the new random addresses to find out which short addresses are existing.
	fb102QueryRandomAddress (bStart := TRUE,
							 nAddress := TO_BYTE(nAddress),
							 eAddressType := Tc3_DALI.E_DALIAddressType.Short,
							 nRandomAddress=> aChangeAddressList[nAddress].nRandomAddress);	
	IF (NOT fb102QueryRandomAddress.bBusy) THEN
		fb102QueryRandomAddress(bStart := FALSE);
		nAddress := nAddress + 1;
		IF (nAddress > 63) THEN 
			nStep := 30;
		END_IF
	END_IF
30:
	// Write the existing short addresses into the table 
	nRow := 0;
	FOR nAddress := 0 TO 63 DO
		IF (aChangeAddressList[nAddress].nRandomAddress > 0) THEN
			aChangeAddressList[nRow].nOldAddress := TO_BYTE(nAddress);
			nRow := nRow + 1;
		END_IF
	END_FOR
	nStep := 40;
40:
	// Hide unused rows in the table
	nHideLine := 0;
	FOR nAddress := 0 TO 63 DO 
		IF (aChangeAddressList[nAddress].nRandomAddress <> 0) THEN
			aShortAddress[nHideLine] := nAddress;
			nHideLine := nHideLine + 1;
		END_IF
	END_FOR	
	FOR nAddress := nHideLine TO 63 DO 
		aNoShortAddress[nAddress] := TRUE;
	END_FOR
	FOR nAddress := 0 TO (nHideLine-1) DO
		aNoShortAddress[nAddress] := FALSE;
	END_FOR	
	aChangeAddressList[nHideLine].nOldAddress := 255;
	FOR nAddress := 0 TO nHideLine DO
		aChangeAddressList[nAddress].nNewAddress := aChangeAddressList[nAddress].nOldAddress;
	END_FOR
	nStep := 0;
{endregion}
60:
{region "Write Changed Addresses"}
	fb102ChangeAddresses(bStart := TRUE,
						 aChangeAddressList := aChangeAddressList);
	IF (NOT fb102ChangeAddresses.bBusy) THEN
		fb102ChangeAddresses(bStart := FALSE,
							 aChangeAddressList := aChangeAddressList);
		nStep := 70;
	END_IF
{endregion}
70:
{region "WriteNewAddressToOldAddress"}
	FOR nAddress := 0 TO 63 DO
		aChangeAddressList[nAddress].nOldAddress := aChangeAddressList[nAddress].nNewAddress;
	END_FOR
	nStep := 0;
{endregion}
END_CASE

END_FUNCTION_BLOCK

// ---- Tc3_DALI_PLC_Commissioning_Tool/POUs/Communication.TcPOU
PROGRAM Communication
VAR_INPUT
END_VAR
VAR
	aKL6821Communication			:	ARRAY [1..GVL_Internal.nNumberOfDALI_Lines] OF FB_KL6821Communication;
	eCommandKBusWatchdog			:	E_DALIConfigurationCommand;
	eCommandDI1RisingEdge			:	E_DALIConfigurationCommand;
	eCommandDI1FallingEdge			:	E_DALIConfigurationCommand;
	eCommandDI2RisingEdge			:	E_DALIConfigurationCommand;
	eCommandDI2FallingEdge			:	E_DALIConfigurationCommand;
	InitTrig						:	R_TRIG;
	nStep							:	INT;
	bInitialize						:	BOOL;
	bDefaultValues					:	BOOL;
	bResetInactiveProcessImage		:	BOOL;
	bDoNotLockProcessImage			:	BOOL;
	bInternalPowerSupplyDisabled	:	BOOL;
	bFirstCycle						:	BOOL := TRUE;
	rTrigInternalPowerSupply		:	R_TRig;
	fTrigInternalPowerSupply		:	f_TRig;
	nTerminal						:	INT := 1;
END_VAR

tc3_DALI.GVL.eEventTraceLevel := TcEventSeverity.Verbose;
IF bFirstCycle THEN
	nStep := 5;
END_IF

InitTrig (CLK := bInitialize);
IF (InitTrig.Q) THEN
	nStep := 10;
END_IF

InitTrig (CLK := bDefaultValues);
IF (InitTrig.Q) THEN
	nStep := 20;
end_if

InitTrig (CLK := bResetInactiveProcessImage);
IF (InitTrig.Q) THEN
	nStep := 30;
END_IF

rTrigInternalPowerSupply (CLK := bInternalPowerSupplyDisabled);
fTrigInternalPowerSupply (CLK := bInternalPowerSupplyDisabled);
IF (rTrigInternalPowerSupply.Q OR fTrigInternalPowerSupply.Q) THEN
	nStep := 40;
END_IF

CASE nStep OF
0:;
5: // Initialization
	FOR nTerminal := 1 TO GVL_Internal.nNumberOfDALI_Lines DO
		eCommandKBusWatchdog := aKL6821Communication[nTerminal].eCommandKBusWatchdog;
		eCommandDI1RisingEdge := aKL6821Communication[nTerminal].eCommandDI1RisingEdge;
		eCommandDI1FallingEdge := aKL6821Communication[nTerminal].eCommandDI1FallingEdge;
		eCommandDI2RisingEdge := aKL6821Communication[nTerminal].eCommandDI2RisingEdge;
		eCommandDI2FallingEdge := aKL6821Communication[nTerminal].eCommandDI2FallingEdge;
		bDoNotLockProcessImage := aKL6821Communication[nTerminal].bDoNotLockProcessImage;
		bInternalPowerSupplyDisabled := aKL6821Communication[nTerminal].bDisableInternalPowerSupply;
	END_FOR
	bFirstCycle := FALSE;
	nStep := 0;
10: // Write changed parameters from visu to specific KL6821
	aKL6821Communication[GVL_Internal.nDALILine].eCommandKBusWatchdog := eCommandKBusWatchdog;
	aKL6821Communication[GVL_Internal.nDALILine].eCommandDI1RisingEdge := eCommandDI1RisingEdge;
	aKL6821Communication[GVL_Internal.nDALILine].eCommandDI1FallingEdge := eCommandDI1FallingEdge;
	aKL6821Communication[GVL_Internal.nDALILine].eCommandDI2RisingEdge := eCommandDI2RisingEdge;
	aKL6821Communication[GVL_Internal.nDALILine].eCommandDI2FallingEdge := eCommandDI2FallingEdge;
	aKL6821Communication[GVL_Internal.nDALILine].bDoNotLockProcessImage := bDoNotLockProcessImage;
	bInitialize := FALSE;
	aKL6821Communication[GVL_Internal.nDALILine].bInitialise := TRUE;
	nStep := 0;
20: // Set default values to specific KL6821 from visu
	eCommandKBusWatchdog := aKL6821Communication[GVL_Internal.nDALILine].eCommandKBusWatchdog := E_DALIConfigurationCommand.DoNothing;
	eCommandDI1RisingEdge := aKL6821Communication[GVL_Internal.nDALILine].eCommandDI1RisingEdge := E_DALIConfigurationCommand.Off;
	eCommandDI1FallingEdge := aKL6821Communication[GVL_Internal.nDALILine].eCommandDI1FallingEdge := E_DALIConfigurationCommand.DoNothing;
	eCommandDI2RisingEdge := aKL6821Communication[GVL_Internal.nDALILine].eCommandDI2RisingEdge := E_DALIConfigurationCommand.RecallMaxLevel;
	eCommandDI2FallingEdge := aKL6821Communication[GVL_Internal.nDALILine].eCommandDI2FallingEdge := E_DALIConfigurationCommand.DoNothing;
	aKL6821Communication[GVL_Internal.nDALILine].bDoNotLockProcessImage := FALSE;
	bDefaultValues := FALSE;
	aKL6821Communication[GVL_Internal.nDALILine].bInitialise := TRUE;
	nStep := 0;
30: // Reset inactive process image on specific Kl6821 from visu
	bResetInactiveProcessImage := FALSE;
	aKL6821Communication[GVL_Internal.nDALILine].bResetInactiveProcessImage := TRUE;
	nStep := 0;
40: // Enable or disable internal power supply of specific KL6821
	aKL6821Communication[GVL_Internal.nDALILine].bDisableInternalPowerSupply := bInternalPowerSupplyDisabled;
	aKL6821Communication[GVL_Internal.nDALILine].bInitialise := TRUE;
	nStep := 0;
END_CASE

FOR nTerminal := 1 TO GVL_Internal.nNumberOfDALI_Lines DO
aKL6821Communication[nTerminal](stInData := GVL.aKL6821InData[nTerminal], stOutData := GVL.aKL6821OutData[nTerminal]);		
END_FOR

IF (NOT aKL6821Communication[GVL_Internal.nDALILine].bInitialising) THEN
	aKL6821Communication[GVL_Internal.nDALILine].bInitialise := FALSE;
END_IF
IF (NOT aKL6821Communication[GVL_Internal.nDALILine].bProcessImageInactive) THEN
	aKL6821Communication[GVL_Internal.nDALILine].bResetInactiveProcessImage := FALSE;
END_IF

END_PROGRAM

// ---- Tc3_DALI_PLC_Commissioning_Tool/POUs/DALI_PLC_Commissioning/FB_Part102Groups.TcPOU
FUNCTION_BLOCK FB_Part102Groups
VAR_INPUT
	ipDALICommunication				:	I_DALICommunication;
END_VAR
VAR_OUTPUT
	bBusy							:	BOOL;
END_VAR
VAR
	{region "Visu"}
	nGroupAddress					:	BYTE;
	bRead							:	BOOL;
	bWrite   						:	BOOL;
	bSwitchOn						:	BOOL;
	bSwitchOff   					:	BOOL;
	aShowAlarmState					:	ARRAY [0..63] OF BOOL;
	aActivateButton					:	ARRAY [0..63] OF BOOL;
	aButtonClick					:	ARRAY [0..63] OF BOOL;
	{endregion}
	i								:	INT;
	bHideWaitSymbol					:	BOOL := TRUE;
	nStep							:	INT;
	nAddress						:	BYTE;
	nNewAddress						:	BYTE;
	fbRecallMaxLevel				:	FB_DALI102RecallMaxLevel(0);
	fbOff							:	FB_DALI102Off(0);
	fb102QueryGroups				:	FB_DALI102QueryGroups(0);
	fb102AddToGroup					:	FB_DALI102AddToGroup(0);
	fb102RemoveFromGroup			:	FB_DALI102RemoveFromGroup(0);
	aDeviceGroupState				:	ARRAY [0..63] OF BYTE; // 0: device isn't present / 1: device belongs to the group / 2: device is not part of the group
END_VAR

{region "Detect Commands"}
IF (bSwitchOn AND (nStep = 0)) THEN
	nStep := 10;
	bSwitchOn := FALSE;
END_IF

IF (bSwitchOff AND (nStep = 0)) THEN
	nStep := 20;
	bSwitchOff := FALSE;
END_IF

IF (bRead AND (nStep = 0)) THEN
	nStep := 1000;
	bRead := FALSE;
	bHideWaitSymbol := FALSE;
	nAddress := 0;
END_IF

IF (bWrite AND (nStep = 0)) THEN
	bWrite := FALSE;
	bHideWaitSymbol := FALSE;
	FOR i := 0 TO 63 DO
		IF (aDeviceGroupState[i] <> 0) THEN
			nAddress := TO_BYTE(i);
			nStep := 2000;
			EXIT;
		 END_IF
	END_FOR
END_IF

IF (nStep = 0) THEN
	FOR i := 0 TO 63 DO
		IF aButtonClick[i] THEN
			aButtonClick[i] := FALSE;
			CASE aDeviceGroupState[i] OF
			1:	// remove device from group
				aActivateButton[i] := TRUE;
				aShowAlarmState[i] := FALSE;
				aDeviceGroupState[i] := 2;
			2:	// add device to group
				aActivateButton[i] := TRUE;
				aShowAlarmState[i] := TRUE;
				aDeviceGroupState[i] := 1;
			ELSE
				aActivateButton[i] := FALSE;
				aShowAlarmState[i] := FALSE;
				aDeviceGroupState[i] := 0;
			END_CASE
		END_IF 
	END_FOR
END_IF
{endregion}
{region "Manage Dialog Selection}
IF (nStep = 0) THEN
	bBusy := FALSE;
ELSE
	bBusy := TRUE;
END_IF
{endregion}
{region "Execute Commands"}
CASE nStep OF
0:
{region "Init"}
	bSwitchOn := FALSE;
	bSwitchOff := FALSE;
	bRead := FALSE;
	bWrite := FALSE;
	bHideWaitSymbol := TRUE;

	fbRecallMaxLevel.ipDALICommunication := ipDALICommunication;
	fbOff.ipDALICommunication := ipDALICommunication;
	fb102QueryGroups.ipDALICommunication := ipDALICommunication;
	fb102AddToGroup.ipDALICommunication := ipDALICommunication;
	fb102RemoveFromGroup.ipDALICommunication := ipDALICommunication;
{endregion}
10:
{region "Recall Max Level"}
	fbRecallMaxLevel(bStart := TRUE,
					 nAddress := nGroupAddress,
					 eAddressType := E_DALIAddressType.Group,
					 eCommandPriority := E_DALICommandPriority.Middle);
	IF (NOT fbRecallMaxLevel.bBusy) THEN
		fbRecallMaxLevel(bStart := FALSE);
		nStep := 0;
	END_IF
{endregion}
20:
{region "Off"}
	fbOff(bStart := TRUE,
		  nAddress := nGroupAddress,
		  eAddressType := E_DALIAddressType.Group,
		  eCommandPriority := E_DALICommandPriority.Middle);
	IF (NOT fbOff.bBusy) THEN
		fbOff(bStart := FALSE);
		nStep := 0;
	END_IF
{endregion}
1000:
{region "Read"}
	fb102QueryGroups(bStart := TRUE,
					 nAddress := nAddress,
					 eAddressType := E_DALIAddressType.Short,
					 eCommandPriority := E_DALICommandPriority.Middle);
	IF (NOT fb102QueryGroups.bBusy) THEN
		IF (NOT fb102QueryGroups.bError) THEN
			IF ((fb102QueryGroups.nGroups AND SHL(16#0001, TO_WORD(nGroupAddress))) <> 0) THEN
				aDeviceGroupState[nAddress] := 1;
			ELSE
				aDeviceGroupState[nAddress] := 2;
			END_IF
		ELSE
			aDeviceGroupState[nAddress] := 0;
		END_IF
		fb102QueryGroups(bStart := FALSE);
		nAddress := nAddress + 1;
		IF (nAddress > 63) THEN
			FOR i := 0 TO 63 DO
				CASE aDeviceGroupState[i] OF
				0:	// device isn't present
					aActivateButton[i] := FALSE;
					aShowAlarmState[i] := FALSE;
				1:	// device belongs to the group
					aActivateButton[i] := TRUE;
					aShowAlarmState[i] := TRUE;
				2:	// device is not part of the group
					aActivateButton[i] := TRUE;
					aShowAlarmState[i] := FALSE;
				ELSE
					aActivateButton[i] := FALSE;
					aShowAlarmState[i] := FALSE;
				END_CASE
			END_FOR
			nStep := 0;
		END_IF
	END_IF
{endregion}
2000:
{region "Write"}
	IF (aDeviceGroupState[nAddress] = 1) THEN
		// add to group
		fb102AddToGroup(bStart := TRUE,
						nAddress := nAddress,
						eAddressType := E_DALIAddressType.Short,
						eCommandPriority := E_DALICommandPriority.Middle,
						nGroup := nGroupAddress);
		IF (NOT fb102AddToGroup.bBusy) THEN
			fb102AddToGroup(bStart := FALSE);
			nStep := 2010;
		END_IF
	ELSIF  (aDeviceGroupState[nAddress] = 2) THEN
		// remove group
		fb102RemoveFromGroup(bStart := TRUE,
							 nAddress := nAddress,
							 eAddressType := E_DALIAddressType.Short,
							 eCommandPriority := E_DALICommandPriority.Middle,
							 nGroup := nGroupAddress);
		IF (NOT fb102RemoveFromGroup.bBusy) THEN
			fb102RemoveFromGroup(bStart := FALSE);
			nStep := 2010;
		END_IF
	ELSE
		nStep := 2010;
	END_IF
2010:
	FOR i := (nAddress + 1) TO 63 DO
		IF (aDeviceGroupState[i] <> 0) THEN
			nNewAddress := TO_BYTE(i);
			nStep := 2000;
			EXIT;
		 END_IF
	END_FOR
	IF (nAddress = nNewAddress) THEN
		nStep := 0;
	ELSE
		nAddress := nNewAddress;
		nStep := 2000;
	END_IF
{endregion}
	ELSE
		nStep := 0;
END_CASE
{endregion}

END_FUNCTION_BLOCK

// ---- Tc3_DALI_PLC_Commissioning_Tool/POUs/DALI_PLC_Commissioning/FB_Part102Parameters.TcPOU
FUNCTION_BLOCK FB_Part102Parameters
VAR_INPUT
	ipDALICommunication				:	I_DALICommunication;
END_VAR
VAR_OUTPUT
	bBusy							:	BOOL;
END_VAR
VAR
	{region "Visu"}
	nAddressRange					:	BYTE; // 0: single short address / 1: address range
	nStartAddress					:	BYTE;
	nEndAddress						:	BYTE;
	nSelectedAddress				:	INT := 255;
	bRead							:	BOOL;
	bWrite							:	BOOL;
	bHideWaitSymbol					:	BOOL := TRUE;
	aParameters						:	ARRAY [0..63] OF ST_DALI102Parameters;
	{endregion}
	i								:	INT;
	nStep							:	INT;
	nAddress						:	BYTE;
	fb102QueryActualLevel			:	FB_DALI102QueryActualLevel(0);
	fb102QueryMinLevel				:	FB_DALI102QueryMinLevel(0);
	fb102QueryMaxLevel				:	FB_DALI102QueryMaxLevel(0);
	fb102QueryFadeTimeFadeRate		:	FB_DALI102QueryFadeTimeFadeRate(0);
	fb102QueryPowerOnLevel			: 	FB_DALI102QueryPowerOnLevel(0);
	fb102QuerySystemFailureLevel  	: 	FB_DALI102QuerySystemFailureLevel(0);
	fb102QueryPhysicalMinimum		: 	FB_DALI102QueryPhysicalMinimum(0); 
	fb102QueryDeviceTypes			: 	FB_DALI102QueryDeviceTypes(0);

	fb102DirectArcPowerControl		:	FB_DALI102DirectArcPowerControl(0);
	fb102SetMinLevel				:	FB_DALI102SetMinLevel(0);
	fb102SetMaxLevel				:	FB_DALI102SetMaxLevel(0);
	fb102SetFadeTime				:	FB_DALI102SetFadeTime(0);
	fb102SetFadeRate				:	FB_DALI102SetFadeRate(0);
	fb102SetPowerOnLevel			: 	FB_DALI102SetPowerOnLevel(0);
	fb102SetSystemFailureLevel  	: 	FB_DALI102SetSystemFailureLevel(0);
END_VAR

{region "Detect Commands"}
IF (bRead AND (nStep = 0)) THEN
	nStep := 10;
	bRead := FALSE;
	bHideWaitSymbol := FALSE;
	IF (nAddressRange = 0) THEN // single short address
		nAddress := TO_BYTE(nSelectedAddress);
	ELSIF (nAddressRange = 1) THEN // address range
		nAddress := nStartAddress;
	END_IF
END_IF

IF (bWrite AND (nStep = 0)) THEN
	nStep := 1000;
	bWrite := FALSE;
	bHideWaitSymbol := FALSE;
	IF (nAddressRange = 0) THEN
		nAddress := TO_BYTE(nSelectedAddress);
	END_IF
END_IF
{endregion}
{region "Avoid errors in line output"}
IF (nSelectedAddress < 0) THEN
	nSelectedAddress := 255;
END_IF
{endregion}
{region "Manage Dialog Selection}
IF (nStep = 0) THEN
	bBusy := FALSE;
ELSE
	bBusy := TRUE;
END_IF
{endregion}
{region "Execute Commands"}
CASE nStep OF
0:
{region "Init"}
	bRead := FALSE;
	bWrite := FALSE;
	bHideWaitSymbol := TRUE;

	fb102QueryActualLevel.ipDALICommunication := ipDALICommunication;
	fb102QueryMinLevel.ipDALICommunication := ipDALICommunication;
	fb102QueryMaxLevel.ipDALICommunication := ipDALICommunication;
	fb102QueryFadeTimeFadeRate.ipDALICommunication := ipDALICommunication;
	fb102QueryPowerOnLevel.ipDALICommunication := ipDALICommunication;
	fb102QuerySystemFailureLevel.ipDALICommunication := ipDALICommunication;
	fb102QueryPhysicalMinimum.ipDALICommunication := ipDALICommunication;
	fb102QueryDeviceTypes.ipDALICommunication := ipDALICommunication;
	fb102DirectArcPowerControl.ipDALICommunication := ipDALICommunication;
	fb102SetMinLevel.ipDALICommunication := ipDALICommunication;
	fb102SetMaxLevel.ipDALICommunication := ipDALICommunication;
	fb102SetFadeTime.ipDALICommunication := ipDALICommunication;
	fb102SetFadeRate.ipDALICommunication := ipDALICommunication;
	fb102SetPowerOnLevel.ipDALICommunication := ipDALICommunication;
	fb102SetSystemFailureLevel.ipDALICommunication := ipDALICommunication;
{endregion}
{region "Read"}
10:
{region "Query Actual Level"}
	fb102QueryActualLevel(bStart := TRUE,
						  nAddress := nAddress,
						  eAddressType := E_DALIAddressType.Short,
						  eCommandPriority := E_DALICommandPriority.Middle);
	IF (NOT fb102QueryActualLevel.bBusy) THEN
		nStep := 20;
		fb102QueryActualLevel(bStart := FALSE);
		IF (NOT fb102QueryActualLevel.bError) THEN
			aParameters[nAddress].nActualLevel := fb102QueryActualLevel.nActualLevel;
		END_IF

		IF (fb102QueryActualLevel.ipResultMessage.nEventId = TC_EVENTS.TcDALIEventClass.NoResponseFromTheDALIDevice.nEventId) THEN 
			aParameters[nAddress].nActualLevel := 0;
			aParameters[nAddress].eFadeRate := 255;
			aParameters[nAddress].eFadeTime := 255;
			aParameters[nAddress].nMaxLevel := 0;
			aParameters[nAddress].nMinLevel := 0;
			aParameters[nAddress].nPhysicalMinimum := 0;
			aParameters[nAddress].nPowerOnLevel := 0;
			aParameters[nAddress].nSystemFailureLevel := 0;
			aParameters[nAddress].sDeviceTypes := '';
			IF (nAddressRange = 1) THEN
				nAddress := nAddress+1;
				IF (nAddress <= nEndAddress) THEN
					nStep := 10;
				ELSE
					nStep := 0;
				END_IF
			ELSE 
				nStep := 0;
			END_IF
		END_IF
	END_IF
{endregion}
20:
{region "Query Min Level"}
	fb102QueryMinLevel(bStart := TRUE,
					   nAddress := nAddress,
					   eAddressType := E_DALIAddressType.Short,
					   eCommandPriority := E_DALICommandPriority.Middle);
	IF (NOT fb102QueryMinLevel.bBusy) THEN
		IF (not fb102QueryMinLevel.bError) THEN
			aParameters[nAddress].nMinLevel := fb102QueryMinLevel.nMinLevel;
		END_IF
		fb102QueryMinLevel(bStart := FALSE);
		nStep := 30;
	END_IF
{endregion}
30:
{region "Query Max Level"}
	fb102QueryMaxLevel(bStart := TRUE,
					   nAddress := nAddress,
					   eAddressType := E_DALIAddressType.Short,
					   eCommandPriority := E_DALICommandPriority.Middle);
	IF (NOT fb102QueryMaxLevel.bBusy) THEN
		IF (NOT fb102QueryMaxLevel.bError) THEN
			aParameters[nAddress].nMaxLevel := fb102QueryMaxLevel.nMaxLevel;
		END_IF
		fb102QueryMaxLevel(bStart := FALSE);
		nStep := 40;
	END_IF
{endregion}
40:
{region "Query Fade Time Fade Rate"}
	fb102QueryFadeTimeFadeRate(bStart := TRUE,
							   nAddress := nAddress,
							   eAddressType := E_DALIAddressType.Short,
							   eCommandPriority := E_DALICommandPriority.Middle);
	IF (NOT fb102QueryFadeTimeFadeRate.bBusy) THEN
		IF(NOT fb102QueryFadeTimeFadeRate.bError) THEN
			aParameters[nAddress].eFadeRate := fb102QueryFadeTimeFadeRate.eFadeRate;
			aParameters[nAddress].eFadeTime := fb102QueryFadeTimeFadeRate.eFadeTime;
		END_IF
		fb102QueryFadeTimeFadeRate(bStart := FALSE);
		nStep := 50;
	END_IF
{endregion}
50:
{region "Query PowerOn Level"}
	fb102QueryPowerOnLevel(bStart := TRUE,
						   nAddress := nAddress,
						   eAddressType := E_DALIAddressType.Short,
						   eCommandPriority := E_DALICommandPriority.Middle);
	IF (NOT fb102QueryPowerOnLevel.bBusy) THEN
		IF (NOT fb102QueryPowerOnLevel.bError) THEN
			aParameters[nAddress].nPowerOnLevel := fb102QueryPowerOnLevel.nPowerOnLevel;
		END_IF
		fb102QueryPowerOnLevel(bStart := FALSE);
		nStep := 60;
	END_IF
{endregion}
60:
{region "Query System Failure Level"}
	fb102QuerySystemFailureLevel(bStart := TRUE,
								 nAddress := nAddress,
								 eAddressType := E_DALIAddressType.Short,
								 eCommandPriority := E_DALICommandPriority.Middle);
	IF (NOT fb102QuerySystemFailureLevel.bBusy) THEN
		IF (NOT fb102QuerySystemFailureLevel.bError) THEN
			aParameters[nAddress].nSystemFailureLevel := fb102QuerySystemFailureLevel.nSystemFailureLevel;
		END_IF
		fb102QuerySystemFailureLevel(bStart := FALSE);
		nStep := 70;
	END_IF
{endregion}
70:
{region "Query Physical Minimum"}
	fb102QueryPhysicalMinimum(bStart := TRUE,
							  nAddress := nAddress,
							  eAddressType := E_DALIAddressType.Short,
							  eCommandPriority := E_DALICommandPriority.Middle);
	IF (NOT fb102QueryPhysicalMinimum.bBusy) THEN
		IF (NOT fb102QueryPhysicalMinimum.bError) THEN
			aParameters[nAddress].nPhysicalMinimum := fb102QueryPhysicalMinimum.nPhysicalMinimum;
		END_IF
		fb102QueryPhysicalMinimum(bStart := FALSE);
		nStep := 80;
	END_IF
{endregion}
80:
{region "Query Device Types"}
	fb102QueryDeviceTypes(bStart := TRUE,
						  nAddress := nAddress,
						  eAddressType := E_DALIAddressType.Short,
						  eCommandPriority := E_DALICommandPriority.Middle);
	IF (NOT fb102QueryDeviceTypes.bBusy) THEN
		fb102QueryDeviceTypes(bStart := FALSE);
		IF ( NOT fb102QueryDeviceTypes.bError) THEN
			aParameters[nAddress].sDeviceTypes := '';
			FOR i := 1 TO 20 DO
				IF (fb102QueryDeviceTypes.aDeviceTypes[i] > 0) THEN
					IF (fb102QueryDeviceTypes.aDeviceTypes[i] <> 255) THEN
						IF (aParameters[nAddress].sDeviceTypes <> '') THEN
							aParameters[nAddress].sDeviceTypes := CONCAT(aParameters[nAddress].sDeviceTypes, ', ');
						END_IF
						aParameters[nAddress].sDeviceTypes := CONCAT(aParameters[nAddress].sDeviceTypes, TO_STRING(TO_INT(fb102QueryDeviceTypes.aDeviceTypes[i])));
					END_IF
				END_IF
			END_FOR
		END_IF
		IF (nAddressRange = 1) THEN // address range
			nAddress := nAddress + 1;
			IF (nAddress <= nEndAddress) THEN
				nStep := 10;
			ELSE
				nStep := 0;
			END_IF
		ELSE
			nStep := 0;
		END_IF
	END_IF
{endregion}
{endregion}
{region "Write"}
1000:
{region "Direct Arc Power Control"}
	fb102DirectArcPowerControl(bStart := TRUE,
							   nAddress := nAddress,
							   eAddressType := E_DALIAddressType.Short,
							   eCommandPriority := E_DALICommandPriority.Middle,
							   nArcPowerLevel := aParameters[nAddress].nActualLevel);
	IF (NOT fb102DirectArcPowerControl.bBusy) THEN
		fb102DirectArcPowerControl(bStart := FALSE);
		nStep := 1010;
	END_IF
{endregion}
1010:
{region "Set Min Level"}
	fb102SetMinLevel(bStart := TRUE,
					 nAddress := nAddress,
					 eAddressType := E_DALIAddressType.Short,
					 eCommandPriority := E_DALICommandPriority.Middle,
					 nMinLevel := aParameters[nAddress].nMinLevel);
	IF (NOT fb102SetMinLevel.bBusy) THEN
		fb102SetMinLevel(bStart := FALSE);
		nStep := 1020;
	END_IF
{endregion}
1020:
{region "Set Max Level"}
	fb102SetMaxLevel(bStart := TRUE,
					 nAddress := nAddress,
					 eAddressType := E_DALIAddressType.Short,
					 eCommandPriority := E_DALICommandPriority.Middle,
					 nMaxLevel := aParameters[nAddress].nMaxLevel);
	IF (NOT fb102SetMaxLevel.bBusy) THEN
		fb102SetMaxLevel(bStart := FALSE);
		nStep := 1030;
	END_IF
{endregion}
1030:
{region "Set Fade Time"}
	fb102SetFadeTime(bStart := TRUE,
					 nAddress := nAddress,
					 eAddressType := E_DALIAddressType.Short,
					 eCommandPriority := E_DALICommandPriority.Middle,
					 eFadeTime := aParameters[nAddress].eFadeTime);
	IF (NOT fb102SetFadeTime.bBusy) THEN
		fb102SetFadeTime(bStart := FALSE);
		nStep := 1040;
	END_IF
{endregion}
1040:
{region "Set Fade Rate"}
	fb102SetFadeRate(bStart := TRUE,
					 nAddress := nAddress,
					 eAddressType := E_DALIAddressType.Short,
					 eCommandPriority := E_DALICommandPriority.Middle,
					 eFadeRate := aParameters[nAddress].eFadeRate);
	IF (NOT fb102SetFadeRate.bBusy) THEN
		fb102SetFadeRate(bStart := FALSE);
		nStep := 1050;
	END_IF
{endregion}
1050:
{region "Set Power On Level"}
	fb102SetPowerOnLevel(bStart := TRUE,
						 nAddress := nAddress,
						 eAddressType := E_DALIAddressType.Short,
						 eCommandPriority := E_DALICommandPriority.Middle,
						 nPowerOnLevel := aParameters[nAddress].nPowerOnLevel);
	IF (NOT fb102SetPowerOnLevel.bBusy) THEN
		fb102SetPowerOnLevel(bStart := FALSE);
		nStep := 1060;
	END_IF
{endregion}
1060:
{region "Set System Failure Level"}
	fb102SetSystemFailureLevel(bStart := TRUE,
							   nAddress := nAddress,
							   eAddressType := E_DALIAddressType.Short,
							   eCommandPriority := E_DALICommandPriority.Middle,
							   nSystemFailureLevel := aParameters[nAddress].nSystemFailureLevel);
	IF (NOT fb102SetSystemFailureLevel.bBusy) THEN
		fb102SetSystemFailureLevel(bStart := FALSE);
		IF (nAddressRange = 1) THEN // address range
			nAddress := nAddress + 1;
			IF (nAddress <= nEndAddress) THEN
				nStep := 1000;
			ELSE
				nStep := 0;
			END_IF
		ELSE
			nStep := 0;
		END_IF
	END_IF
{endregion}
ELSE
	nStep := 0;
END_CASE
{endregion}

END_FUNCTION_BLOCK

// ---- Tc3_DALI_PLC_Commissioning_Tool/POUs/DALI_PLC_Commissioning/FB_Part102Scenes.TcPOU
FUNCTION_BLOCK FB_Part102Scenes
VAR_INPUT
	ipDALICommunication		:	I_DALICommunication;
END_VAR
VAR_OUTPUT
	bBusy					:	BOOL;
END_VAR
VAR
	{region "Visu"}
	nScene					:	BYTE;
	bGoToScene				:	BOOL;
	bSwitchOff				:	BOOL;
	bRead					:	BOOL;
	bWrite		 			:	BOOL;
	aScene					:	ARRAY [0..63] OF BYTE;
	aNoShortAddress			:	ARRAY [0..63] OF BOOL;
	bHideWaitSymbol			:	BOOL := TRUE;
	{endregion}
	nStep					:	INT; // Running index
	nAddress				:	INT;
	aFont					:	ARRAY [0..63] OF DWORD;

	fb102QuerySceneLevel	:	FB_DALI102QuerySceneLevel(0);
	fb102SetScene			:	FB_DALI102SetScene(0);
	fb102GoToScene			:	FB_DALI102GoToScene(0);
	fb102Off				:	FB_DALI102Off(0);
END_VAR

{region "Detect Commands"}
IF (bRead AND (nStep = 0)) THEN 
	nStep := 10;
	bRead := FALSE;
	bHideWaitSymbol := FALSE;
END_IF

IF (bWrite AND (nStep = 0)) THEN 
	nStep := 20;
	bWrite := FALSE;
	bHideWaitSymbol := FALSE;
END_IF

IF (bGoToScene AND (nStep = 0)) THEN 
	nStep := 30;
	bGoToScene := FALSE;
	bHideWaitSymbol := FALSE;
END_IF

IF (bSwitchOff AND (nStep = 0)) THEN
	nStep := 40;
	bSwitchOff := FALSE;
	bHideWaitSymbol := FALSE;
END_IF
{endregion}
{region "Manage Dialog Selection}
IF (nStep = 0) THEN
	bBusy := FALSE;
ELSE
	bBusy := TRUE;
END_IF
{endregion}
{region "Execute Commands"}
CASE nStep OF
0:
{region "Init"}
	bRead := FALSE;	
	bWrite := FALSE;
	bGoToScene := FALSE;
	bSwitchOff := FALSE;
	bHideWaitSymbol := TRUE;
	nAddress := 0;

	fb102QuerySceneLevel.ipDALICommunication := ipDALICommunication;
	fb102SetScene.ipDALICommunication := ipDALICommunication;
	fb102GoToScene.ipDALICommunication := ipDALICommunication;
	fb102Off.ipDALICommunication := ipDALICommunication;
{endregion}
10:
{region "Query Scene Level"}
	fb102QuerySceneLevel(bStart := TRUE, 
						 nAddress := TO_BYTE(nAddress),
						 eAddressType := Tc3_DALI.E_DALIAddressType.Short,
						 eCommandPriority := Tc3_DALI.E_DALICommandPriority.Middle,
						 nScene := nScene,
						 nSceneLevel=> aScene[nAddress]);
	IF (NOT fb102QuerySceneLevel.bBusy) THEN
		fb102QuerySceneLevel (bStart:= FALSE);
		IF (fb102QuerySceneLevel.ipResultMessage.nEventId = TC_EVENTS.TcDALIEventClass.NoResponseFromTheDALIDevice.nEventId) THEN // Deletes not existing short addresses from display
			aNoShortAddress[nAddress] := TRUE;
			aFont[nAddress] := 16#FF505050;
		ELSE
			aNoShortAddress[nAddress] := FALSE;
			aFont[nAddress] := 16#FFFFFFFF;
		END_IF
		nAddress := nAddress + 1;
		IF (nAddress > 63)THEN
			nStep := 0;
		END_IF
	END_IF
{endregion}
20:
{region "Set Scene"}
	IF (aNoShortAddress[nAddress] = TRUE) THEN
		nAddress := nAddress + 1;
		IF (nAddress > 63)THEN
			nStep := 0;
		END_IF
	ELSE
		fb102SetScene(bStart := TRUE,
					  nAddress := TO_BYTE(nAddress),
					  eAddressType := Tc3_DALI.E_DALIAddressType.Short,
					  eCommandPriority := Tc3_DALI.E_DALICommandPriority.Middle,
					  nSceneLevel := aScene[nAddress],
					  nScene := nScene);
		IF (NOT fb102SetScene.bBusy) THEN
			fb102SetScene(bStart := FALSE);
			nAddress := nAddress + 1;
			IF (nAddress > 63)THEN
				nStep := 0;
			END_IF
		END_IF
	END_IF
{endregion}
30:
{region "Go To Scene"}
	IF (aNoShortAddress[nAddress] = TRUE) THEN
		nAddress := nAddress + 1;
		IF (nAddress > 63)THEN
			nStep := 0;
		END_IF
	ELSE
		fb102GoToScene(bStart := TRUE,
					   nAddress := TO_BYTE(nAddress),
					   eAddressType := Tc3_DALI.E_DALIAddressType.Short,
					   eCommandPriority := Tc3_DALI.E_DALICommandPriority.Middle,
					   nScene := nScene);
		IF (NOT fb102GoToScene.bBusy) THEN
			fb102GoToScene(bStart := FALSE);
			nAddress := nAddress + 1;
			IF (nAddress > 63)THEN
				nStep := 0;
			END_IF
		END_IF
	END_IF
{endregion}
40:
{region "Switch Off"}
	fb102Off(bStart := TRUE,
			 nAddress := TO_BYTE(nAddress),
			 eAddressType := Tc3_DALI.E_DALIAddressType.Broadcast,
			 eCommandPriority := Tc3_DALI.E_DALICommandPriority.Middle);
	IF (NOT fb102Off.bBusy) THEN
		fb102Off(bStart := FALSE);
		nStep := 0;
	END_IF
{endregion}
END_CASE
{endregion}

END_FUNCTION_BLOCK

// ---- Tc3_DALI_PLC_Commissioning_Tool/POUs/DALI_PLC_Commissioning/FB_Part103Addressing.TcPOU
FUNCTION_BLOCK FB_Part103Addressing
VAR_INPUT
	ipDALICommunication			:	I_DALICommunication;
END_VAR
VAR_OUTPUT
	bBusy						:	BOOL;
END_VAR
VAR
	{region "Visu"}
	bScanDevices				:	BOOL;
	bStartChangeAddress			:	BOOL;
	bStartRandomAddressing		:	BOOL;
	nStartAddress				:	BYTE;
	bNewInstallation			:	BOOL;
	bOpticalFeedback			:	BOOL;
	bHideWaitSymbol				:	BOOL := TRUE;
	{endregion}
	nStep						:	INT;
	nAddress					:	INT;
	aChangeAddressList			:	ARRAY [0..63] OF ST_DALIChangeAddressList;
	aShortAddress				:	ARRAY [0..63] OF INT;
	aNoShortAddress				:	ARRAY [0..63] OF BOOL;
	nRow						:	INT;
	nHideLine					:	INT; // Variable to find out how many rows are used

	fb103Addressing				:	FB_DALI103Addressing(0);
	fb103QueryRandomAddress		:	FB_DALI103QueryRandomAddress(0);
	fb103ChangeAddresses		:	FB_DALI103ChangeAddresses(0);
END_VAR

{region "Detect Commands"}
IF (bStartRandomAddressing AND (nStep = 0)) THEN
	nStep := 10;
	bStartRandomAddressing := FALSE;
	bHideWaitSymbol := FALSE;
END_IF

IF (bScanDevices AND (nStep = 0)) THEN
	nStep := 20;
	nAddress:=0; 
	bScanDevices := FALSE;
	bHideWaitSymbol := FALSE;
END_IF

IF (bStartChangeAddress AND (nStep = 0)) THEN
	nStep := 60;
	bStartChangeAddress := FALSE;
	bHideWaitSymbol := FALSE;
END_IF
{endregion}
{region "Manage Dialog Selection}
IF (nStep = 0) THEN
	bBusy := FALSE;
ELSE
	bBusy := TRUE;
END_IF
{endregion}	 
{region "Execute Commands"}
CASE nStep OF
0:
{region "Init"}
	bScanDevices := FALSE;
	bStartChangeAddress := FALSE;
	bStartRandomAddressing := FALSE;
	bHideWaitSymbol := TRUE;

	fb103Addressing.ipDALICommunication := ipDALICommunication;
	fb103QueryRandomAddress.ipDALICommunication := ipDALICommunication;
	fb103ChangeAddresses.ipDALICommunication := ipDALICommunication;
{endregion}
10:
{region "RandomAddressing"}
	fb103Addressing.nOptions := 0;

	IF bNewInstallation THEN
		fb103Addressing.nOptions := fb103Addressing.nOptions OR Tc3_DALI.GVL.cCompleteNewInstallation;
	END_IF

	IF bOpticalFeedback THEN
		fb103Addressing.nOptions := fb103Addressing.nOptions OR Tc3_DALI.GVL.cOpticalFeedback;
	END_IF

	fb103Addressing(bStart := TRUE,
					nStartWithShortAddress := nStartAddress);
	IF (NOT fb103Addressing.bBusy) THEN
		fb103Addressing(bStart := FALSE);
		nStep := 0;	
	END_IF
{endregion}
{region "Read Existing Addresses"}
20:
	// Query of the new random addresses to find out which short addresses are existing.
	fb103QueryRandomAddress (bStart := TRUE,
							 nAddress := TO_BYTE(nAddress),
							 eAddressType := Tc3_DALI.E_DALIAddressType.Short,
							 nRandomAddress=> aChangeAddressList[nAddress].nRandomAddress);
	IF (NOT fb103QueryRandomAddress.bBusy) THEN
		fb103QueryRandomAddress(bStart := FALSE);
		nAddress := nAddress + 1;
		IF (nAddress > 63) THEN
			nStep := 30;
		END_IF
	END_IF
30:
	// Write the existing short addresses into the table 
	nRow := 0;
	FOR nAddress := 0 TO 63 DO
		IF (aChangeAddressList[nAddress].nRandomAddress > 0) THEN
			aChangeAddressList[nRow].nOldAddress := TO_BYTE(nAddress);
			nRow := nRow + 1;
		END_IF
	END_FOR
	nStep := 40;
40:
	// Hide unused rows in the table
	nHideLine := 0;
	FOR nAddress := 0 TO 63 DO 
		IF (aChangeAddressList[nAddress].nRandomAddress <> 0) THEN
			aShortAddress[nHideLine] := nAddress;
			nHideLine := nHideLine + 1;
		END_IF
	END_FOR
	FOR nAddress := nHideLine TO 63 DO 
		aNoShortAddress[nAddress] := TRUE;
	END_FOR
	FOR nAddress := 0 TO (nHideLine - 1) DO
		aNoShortAddress[nAddress] := FALSE;
	END_FOR
	aChangeAddressList[nHideLine].nOldAddress := 255;
	FOR nAddress := 0 TO nHideLine DO
		aChangeAddressList[nAddress].nNewAddress := aChangeAddressList[nAddress].nOldAddress;
	END_FOR
	nStep := 0;
{endregion}
60:
{region "Write Changed Addresses}
	fb103ChangeAddresses(bStart := TRUE,
						 aChangeAddressList := aChangeAddressList);
	IF (NOT fb103ChangeAddresses.bBusy) THEN
		fb103ChangeAddresses(bStart := FALSE,
							 aChangeAddressList := aChangeAddressList);
		nStep := 70;
	END_IF
{endregion}
70:
{region "Write New Address To Old Address}
	FOR nAddress := 0 TO 63 DO
		aChangeAddressList[nAddress].nOldAddress := aChangeAddressList[nAddress].nNewAddress;
	END_FOR
	nStep := 0;
{endregion}
END_CASE

END_FUNCTION_BLOCK

// ---- Tc3_DALI_PLC_Commissioning_Tool/POUs/DALI_PLC_Commissioning/FB_Part103Parameters.TcPOU
FUNCTION_BLOCK FB_Part103Parameters
VAR_INPUT
	ipDALICommunication				:	I_DALICommunication;
END_VAR
VAR_OUTPUT
	bBusy							:	BOOL;
END_VAR
VAR
	{region "Visu"}
	nAddressRange					:	BYTE; // 0: single short address / 1: address range
	nStartAddress					:	BYTE;
	nEndAddress						:	BYTE;
	nSelectedAddress				:	INT := 255;
	bRead							:	BOOL;
	bWrite							:	BOOL;
	bHideWaitSymbol					:	BOOL := TRUE;
	aParameters						:	ARRAY [0..63] OF ST_DALI103Parameters;
	{endregion}
	i								:	INT;
	nStep							:	INT;
	nAddress						:	BYTE;
	nInstanceAddress				:	BYTE;
	aNumberOfInstances				:	ARRAY [0..63] OF BYTE;
	aInstance						:	ARRAY [0..63, 0..31] OF BYTE; // First field in array includes short address and second field includes instance type of the according short address.
	bFirstCycle0					:	BOOL;
	bFirstCycle1					:	BOOL;
	bFirstCycle2					:	BOOL;
	bFirstCycle3					:	BOOL;
	bFirstCycle4					:	BOOL;
	nType0							:	INT;
	nType1							:	INT;
	nType2							:	INT;
	nType3							:	INT;
	nType4							:	INT;
	aStringType0					:	ARRAY [0..31] OF STRING;
	aStringType1					:	ARRAY [0..31] OF STRING;
	aStringType2					:	ARRAY [0..31] OF STRING;
	aStringType3					:	ARRAY [0..31] OF STRING;
	aStringType4					:	ARRAY [0..31] OF STRING;

	fb103StartQuiescentMode			:	FB_DALI103StartQuiescentMode(0);
	fb103StopQuiescentMode			:	FB_DALI103StopQuiescentMode(0);
	fb103QueryOperatingMode			:	FB_DALI103QueryOperatingMode(0);
	fb103SetOperatingMode			:	FB_DALI103SetOperatingMode(0);
	fb103QueryNumberOfInstances		:	FB_DALI103QueryNumberOfInstances(0);
	fb103QueryInstanceType			:	FB_DALI103QueryInstanceType(0);
END_VAR

{region "Detect Commands"}
IF (bRead AND (nStep = 0)) THEN
	nStep := 5;
	bRead := FALSE;
	bHideWaitSymbol := FALSE;
	IF (nAddressRange = 0) THEN // single short address
		nAddress := TO_BYTE(nSelectedAddress);
	ELSIF (nAddressRange = 1) THEN // address range
		nAddress := nStartAddress;
	END_IF
END_IF

IF (bWrite AND (nStep = 0)) THEN
	nStep := 1000;
	bWrite := FALSE;
	bHideWaitSymbol := FALSE;
	IF (nAddressRange = 0) THEN
		nAddress := TO_BYTE(nSelectedAddress);
	ELSIF (nAddressRange = 1) THEN // address range
		nAddress := nStartAddress;
	END_IF
END_IF
{endregion}

{region "Avoid errors in line output"}
IF (nSelectedAddress < 0) THEN
	nSelectedAddress := 255;
END_IF
{endregion}

{region "Manage Dialog Selection}
IF (nStep = 0) THEN
	bBusy := FALSE;
ELSE
	bBusy := TRUE;
END_IF
{endregion}

{region "Execute Commands"}
CASE nStep OF
0:
{region "Init"}
	bRead := FALSE;
	bWrite := FALSE;
	bHideWaitSymbol := TRUE;
	fb103StartQuiescentMode.ipDALICommunication := ipDALICommunication;
	fb103StopQuiescentMode.ipDALICommunication := ipDALICommunication;
	fb103QueryOperatingMode.ipDALICommunication := ipDALICommunication;
	fb103SetOperatingMode.ipDALICommunication := ipDALICommunication;
	fb103QueryNumberOfInstances.ipDALICommunication := ipDALICommunication;
	fb103QueryInstanceType.ipDALICommunication := ipDALICommunication;
{endregion}
{region "Read"}
5:
{region "Start Qiescent Mode"}
	fb103StartQuiescentMode(bStart:= TRUE,
							nAddress:= nAddress,
							eAddressType:= Tc3_DALI.E_DALIAddressType.Short,
							eCommandPriority:= Tc3_DALI.E_DALICommandPriority.Middle);
	IF (NOT fb103StartQuiescentMode.bBusy) THEN
		fb103StartQuiescentMode(	bStart:= FALSE);
		nStep := 10;
	END_IF
{endregion}
10:
{region "Query Operating Mode"}
	 fb103QueryOperatingMode(bStart := TRUE,
							 nAddress := nAddress,
							 eAddressType := E_DALIAddressType.Short,
							 eCommandPriority := E_DALICommandPriority.Middle);
	IF (NOT fb103QueryOperatingMode.bBusy) THEN
		aParameters[nAddress].nOperatingMode := fb103QueryOperatingMode.nOperatingMode;
		nStep := 20;
		fb103QueryOperatingMode(bStart := FALSE);
		IF (fb103QueryOperatingMode.ipResultMessage.nEventId = TC_EVENTS.TcDALIEventClass.NoResponseFromTheDALIDevice.nEventId) THEN
			aParameters[nAddress].nOperatingMode := 0; // deleting old entries in the table 
			aParameters[nAddress].sInstanceType0 := '';
			aParameters[nAddress].sInstanceType1 := '';
			aParameters[nAddress].sInstanceType2 := '';
			aParameters[nAddress].sInstanceType3 := '';
			aParameters[nAddress].sInstanceType4 := '';
			IF (nAddressRange = 1) THEN
				nAddress := nAddress+1;	
				IF (nAddress <= nEndAddress) THEN
					nStep := 10;
				ELSE
					nStep := 0;
				END_IF
			ELSE 
				nStep := 0;
			END_IF
		END_IF
	END_IF
{endregion}
20:
{region "Query Number Of Instances"}
	fb103QueryNumberOfInstances(bStart := TRUE,
								nAddress := nAddress,
								eAddressType := E_DALIAddressType.Short,
								eCommandPriority := E_DALICommandPriority.Middle);
	IF (NOT fb103QueryNumberOfInstances.bBusy) THEN
		aNumberOfInstances[nAddress] := fb103QueryNumberOfInstances.nNumberOfInstances;
		fb103QueryNumberOfInstances(bStart := FALSE);
		nStep := 30;
	END_IF
{endregion}
30:
{region "Query Instance Type"}
	fb103QueryInstanceType(bStart := TRUE,
						   nAddress := nAddress,
						   eAddressType := E_DALIAddressType.Short,
						   nInstanceAddress := nInstanceAddress,
						   eInstanceAddressType := Tc3_DALI.E_DALIInstanceAddressType.InstanceNumber,
						   eCommandPriority := E_DALICommandPriority.Middle,
						   eInstanceType=> aInstance[nAddress, nInstanceAddress]);
		IF (NOT fb103QueryInstanceType.bBusy) THEN
			fb103QueryInstanceType(bStart := FALSE);
			nInstanceAddress := nInstanceAddress+1;
			//***************STRING***************
			aParameters[nAddress].sInstanceType0 := '';
			aParameters[nAddress].sInstanceType1 := '';
			aParameters[nAddress].sInstanceType2 := '';
			aParameters[nAddress].sInstanceType3 := '';
			aParameters[nAddress].sInstanceType4 := '';
			bFirstCycle0 := TRUE;
			bFirstCycle1 := TRUE;
			bFirstCycle2 := TRUE;
			bFirstCycle3 := TRUE;
			bFirstCycle4 := TRUE;
			FOR i := 0 TO aNumberOfInstances[nAddress] DO
				IF (aInstance[nAddress, i] = 0) THEN // Read instance type 0
					nType0 := i;
					IF (NOT bFirstCycle0) THEN
						aParameters[nAddress].sInstanceType0 := CONCAT(aParameters[nAddress].sInstanceType0, ',');
					END_IF
					aStringType0[nType0] := TO_STRING(TO_INT(nType0));
					aParameters[nAddress].sInstanceType0 := CONCAT(aParameters[nAddress].sInstanceType0, aStringType0[nType0]);
					bFirstCycle0 := FALSE;
				END_IF
				IF (aInstance[nAddress, i] = 1) THEN // Read instance type 1
					nType1 := i;
					IF (NOT bFirstCycle1) THEN
						aParameters[nAddress].sInstanceType1 := CONCAT(aParameters[nAddress].sInstanceType1, ',');
					END_IF
					aStringType1[nType1] := TO_STRING(TO_INT(nType1));
					aParameters[nAddress].sInstanceType1 := CONCAT(aParameters[nAddress].sInstanceType1, aStringType1[nType1]);
					bFirstCycle1 := FALSE;
				END_IF	
				IF (aInstance[nAddress, i] = 2) THEN  // Read instance type 2
					nType2 := i;
					IF (NOT bFirstCycle2) THEN
						aParameters[nAddress].sInstanceType2 := CONCAT(aParameters[nAddress].sInstanceType2, ',');
					END_IF
					aStringType2[nType2] := TO_STRING(TO_INT(nType2));
					aParameters[nAddress].sInstanceType2 := CONCAT(aParameters[nAddress].sInstanceType2, aStringType2[nType2]);
					bFirstCycle2 := FALSE;
				END_IF
				IF (aInstance[nAddress, i] = 3) THEN // Read instance type 3
					nType3 := i;
					IF (NOT bFirstCycle3) THEN
						aParameters[nAddress].sInstanceType3 := CONCAT(aParameters[nAddress].sInstanceType3, ',');
					END_IF
					aStringType3[nType3] := TO_STRING(TO_INT(nType3));
					aParameters[nAddress].sInstanceType3 := CONCAT(aParameters[nAddress].sInstanceType3, aStringType3[nType3]);	
					bFirstCycle3 := FALSE;
				END_IF
				IF (aInstance[nAddress, i] = 4) THEN // Read instance type 4
					nType4 := i;
					IF (NOT bFirstCycle4) THEN
						aParameters[nAddress].sInstanceType4 := CONCAT(aParameters[nAddress].sInstanceType4, ',');
					END_IF
					aStringType4[nType4] := TO_STRING(TO_INT(nType4));
					aParameters[nAddress].sInstanceType4 := CONCAT(aParameters[nAddress].sInstanceType4, aStringType4[nType4]);
					bFirstCycle4 := FALSE;
				END_IF
			END_FOR
			//********************************************
			IF (nInstanceAddress > aNumberOfInstances[nAddress]) THEN
				nInstanceAddress := 0;
				nStep  := 0;
				IF (nAddressRange = 1) THEN
					nAddress := nAddress + 1;
					IF (nAddress <= nEndAddress) THEN
						nStep := 10;
					ELSE
						nStep := 40;
					END_IF
				END_IF
			END_IF
		END_IF
{endregion}
40:
{region "Stop Qiescent Mode"}
	fb103StopQuiescentMode(bStart := TRUE,
						   nAddress := nAddress,
						   eAddressType := Tc3_DALI.E_DALIAddressType.Short,
						   eCommandPriority := Tc3_DALI.E_DALICommandPriority.Middle);
	IF (NOT fb103StopQuiescentMode.bBusy) THEN
		fb103StopQuiescentMode(bStart := FALSE);
		nStep := 0;
	END_IF
{endregion}
{endregion}
1000:
{region "Write"}
	fb103SetOperatingMode(bStart := TRUE,
						  nAddress := nAddress,
						  eAddressType := E_DALIAddressType.Short,
						  eCommandPriority := E_DALICommandPriority.Middle,
						  nOperatingMode := aParameters[nAddress].nOperatingMode);
	IF (NOT fb103SetOperatingMode.bBusy) THEN
		fb103SetOperatingMode(bStart := FALSE);
		IF (nAddressRange = 0) THEN
			nStep := 0;
		END_IF
		IF (nAddressRange = 1) THEN
			nAddress := nAddress + 1;
			IF (nAddress > nEndAddress) THEN
				nStep := 0;
				nAddress := 0;
			END_IF
		END_IF
	END_IF
{endregion}
 END_CASE

END_FUNCTION_BLOCK

// ---- Tc3_DALI_PLC_Commissioning_Tool/POUs/DALI_PLC_Commissioning/FB_Part300GenericDevice.TcPOU
FUNCTION_BLOCK FB_Part300GenericDevice
VAR_INPUT
	ipDALICommunication			:	I_DALICommunication;
END_VAR
VAR_OUTPUT
	bBusy						:	BOOL;
END_VAR
VAR
	{region "Visu"}
	nInputValue					:	LWORD;
	nInstanceError				:	BYTE;
	nResolution					:	BYTE;
	eEventScheme				:	E_DALIEventScheme;
	nEventFilter				:	DWORD;
	bRead						:	BOOL;
	bWrite						:	BOOL;
	bEnable						:	BOOL;
	bBit0						:	BOOL;
	bBit1						:	BOOL;
	bBit2						:	BOOL;
	bBit3						:	BOOL;
	bBit4						:	BOOL;
	bBit5						:	BOOL;
	bBit6						:	BOOL;
	bBit7						:	BOOL;
	eEventPriority				:	E_DALIEventPriority := E_DALIEventPriority.Middle;
	bIdentify					: 	BOOL;
	{endregion}
	nStep						:	INT;
	nAddress					:	BYTE;
	nInstanceAddress			:	BYTE;
	bHideWaitSymbol				:	BOOL := TRUE;

	fb103StartQuiescentMode		:	FB_DALI103StartQuiescentMode(0);
	fb103StopQuiescentMode		:	FB_DALI103StopQuiescentMode(0);
	fb103QueryInstanceError		:	FB_DALI103QueryInstanceError(0);
	fb103QueryInstanceStatus	:	FB_DALI103QueryInstanceStatus(0);
	fb103QueryResolution		:	FB_DALI103QueryResolution(0);
	fb103QueryInputValue 		:	FB_DALI103QueryInputValue(0);
	fb103QueryEventScheme 		:	FB_DALI103QueryEventScheme(0);
	fb103QueryEventFilter 		:	FB_DALI103QueryEventFilter(0);
	fb103QueryEventPriority		:	FB_DALI103QueryEventPriority(0);
	fb103EnableInstance 		:	FB_DALI103EnableInstance(0);
	fb103DisableInstance		:	FB_DALI103DisableInstance(0);
	fb103SetEventScheme 		:	FB_DALI103SetEventScheme(0);
	fb103SetEventFilter 		:	FB_DALI103SetEventFilter(0);
	fb103SetEventPriority		:	FB_DALI103SetEventPriority(0);
	fb103IdentifyDevice   		:   FB_DALI103IdentifyDevice(0);
END_VAR

{region "Detect Commands"}
IF (bRead AND (nStep = 0)) THEN
	nStep := 5;
	bRead := FALSE;
	bHideWaitSymbol := FALSE;
END_IF

IF (bWrite AND (nStep = 0)) THEN
	nStep := 1000;
	bWrite := FALSE;
	bHideWaitSymbol := FALSE;
END_IF
	 
IF (bIdentify AND (nStep = 0)) THEN
	 nStep := 2000;
	 bIdentify := FALSE;
END_IF
{endregion}
{region "Manage Dialog Selection}
IF (nStep = 0) THEN
	bBusy := FALSE;
ELSE
	bBusy := TRUE;
END_IF
{endregion}
{region "Execute Commands"}
CASE nStep OF
0:
{region "Init"}
	bRead := FALSE;
	bWrite := FALSE;
	bHideWaitSymbol := TRUE;

	fb103StartQuiescentMode.ipDALICommunication := ipDALICommunication;
	fb103StopQuiescentMode.ipDALICommunication := ipDALICommunication;
	fb103QueryInstanceError.ipDALICommunication := ipDALICommunication;
	fb103QueryInstanceStatus.ipDALICommunication := ipDALICommunication;
	fb103QueryResolution.ipDALICommunication := ipDALICommunication;
	fb103QueryInputValue.ipDALICommunication := ipDALICommunication;
	fb103QueryEventScheme.ipDALICommunication := ipDALICommunication;
	fb103QueryEventFilter.ipDALICommunication := ipDALICommunication;
	fb103QueryEventPriority.ipDALICommunication := ipDALICommunication;
	fb103EnableInstance.ipDALICommunication := ipDALICommunication;
	fb103DisableInstance.ipDALICommunication := ipDALICommunication;
	fb103SetEventScheme.ipDALICommunication := ipDALICommunication;
	fb103SetEventFilter.ipDALICommunication := ipDALICommunication;
	fb103SetEventPriority.ipDALICommunication := ipDALICommunication;
    fb103IdentifyDevice.ipDALICommunication := ipDALICommunication;
{endregion}
{region "Read"}
5:
{region "Start Qiescent Mode"}
	fb103StartQuiescentMode(bStart := TRUE,
							eAddressType := Tc3_DALI.E_DALIAddressType.Broadcast,
							eCommandPriority := Tc3_DALI.E_DALICommandPriority.Middle);
	IF (NOT fb103StartQuiescentMode.bBusy) THEN
		fb103StartQuiescentMode(bStart:= FALSE);
		nStep := 10;
	END_IF
{endregion}
10:
{region "Query Instance Error"}
	fb103QueryInstanceError(bStart := TRUE,
							nAddress := nAddress,
							eAddressType := Tc3_DALI.E_DALIAddressType.Short,
							nInstanceAddress := nInstanceAddress,
							eInstanceAddressType := Tc3_DALI.E_DALIInstanceAddressType.InstanceNumber,
							eCommandPriority := Tc3_DALI.E_DALICommandPriority.Middle,
							nInstanceError=> nInstanceError);
	IF (NOT fb103QueryInstanceError.bBusy) THEN
		fb103QueryInstanceError(bStart:= FALSE);
		nStep := 20;
	END_IF
{endregion}
20:
{region "Query Instance Status"}
	fb103QueryInstanceStatus(bStart:= TRUE,
							 nAddress := nAddress,
							 eAddressType := Tc3_DALI.E_DALIAddressType.Short,
							 nInstanceAddress := nInstanceAddress,
							 eInstanceAddressType := Tc3_DALI.E_DALIInstanceAddressType.InstanceNumber,
							 eCommandPriority := Tc3_DALI.E_DALICommandPriority.Middle);
	IF (NOT fb103QueryInstanceStatus.bBusy) THEN
		fb103QueryInstanceStatus(bStart := FALSE);
		IF (fb103QueryInstanceStatus.nInstanceStatus.1) THEN
			bEnable := TRUE;
		END_IF
		nStep := 30;
	END_IF
30:
{region "Query Resolution"}
	fb103QueryResolution(bStart := TRUE,
						 nAddress := nAddress,
						 eAddressType := Tc3_DALI.E_DALIAddressType.Short,
						 nInstanceAddress := nInstanceAddress,
						 eInstanceAddressType := Tc3_DALI.E_DALIInstanceAddressType.InstanceNumber,
						 eCommandPriority := Tc3_DALI.E_DALICommandPriority.Middle,
						 nResolution=> nResolution);
	IF (NOT fb103QueryResolution.bBusy) THEN
		fb103QueryResolution(bStart:= FALSE);
		nStep := 40;
	END_IF
{endregion}
40:
{region "Query Input Value"}
	fb103QueryInputValue(bStart := TRUE,
						 nAddress := nAddress,
						 eAddressType := Tc3_DALI.E_DALIAddressType.Short,
						 nInstanceAddress := nInstanceAddress,
						 eInstanceAddressType := Tc3_DALI.E_DALIInstanceAddressType.InstanceNumber,
						 eCommandPriority := Tc3_DALI.E_DALICommandPriority.Middle,
						 nResolution := nResolution,
						 nInputValue=> nInputValue);
	IF (NOT fb103QueryInputValue.bBusy) THEN
		fb103QueryInputValue(bStart:= FALSE);
		nStep := 50;
	END_IF
{endregion}
50:
{region "Query Event Scheme"}
	fb103QueryEventScheme(bStart := TRUE,
						  nAddress := nAddress,
						  eAddressType := Tc3_DALI.E_DALIAddressType.Short,
						  nInstanceAddress := nInstanceAddress,
						  eInstanceAddressType := Tc3_DALI.E_DALIInstanceAddressType.InstanceNumber,
						  eCommandPriority := Tc3_DALI.E_DALICommandPriority.Middle,
						  eEventScheme=> eEventScheme);
	IF (NOT fb103QueryEventScheme.bBusy) THEN
		fb103QueryEventScheme(bStart:= FALSE);
		nStep := 60;
	END_IF
{endregion}
60:
{region "Query Event Filter"}
	fb103QueryEventFilter(bStart := TRUE,
						  nAddress := nAddress,
						  eAddressType := Tc3_DALI.E_DALIAddressType.Short,
						  nInstanceAddress := nInstanceAddress,
						  eInstanceAddressType := Tc3_DALI.E_DALIInstanceAddressType.InstanceNumber,
						  eCommandPriority := Tc3_DALI.E_DALICommandPriority.Middle,
						  nEventFilter=> nEventFilter);
	IF (NOT fb103QueryEventFilter.bBusy) THEN
		fb103QueryEventFilter(bStart := FALSE);
		bBit0 := nEventFilter.0;
		bBit1 := nEventFilter.1;
		bBit2 := nEventFilter.2;
		bBit3 := nEventFilter.3;
		bBit4 := nEventFilter.4;
		bBit5 := nEventFilter.5;
		bBit6 := nEventFilter.6;
		bBit7 := nEventFilter.7;
		nStep := 90;
	END_IF
{endregion}
90:
{region "Query Event Priority"}
	fb103QueryEventPriority(bStart := TRUE,
							nAddress := nAddress,
							eAddressType := Tc3_DALI.E_DALIAddressType.Short,
							nInstanceAddress := nInstanceAddress,
							eInstanceAddressType := Tc3_DALI.E_DALIInstanceAddressType.InstanceNumber,
							eCommandPriority := Tc3_DALI.E_DALICommandPriority.Middle,
							eEventPriority=> eEventPriority);
	IF (NOT fb103QueryEventPriority.bBusy) THEN
		fb103QueryEventPriority(bStart := FALSE);
		nStep := 100;
	END_IF 
{endregion}
100:
{region "Stop Qiescent Mode"}
	fb103StopQuiescentMode(bStart:= TRUE,
						   eAddressType:= Tc3_DALI.E_DALIAddressType.Broadcast,
						   eCommandPriority:= Tc3_DALI.E_DALICommandPriority.Middle);
	IF (NOT fb103StopQuiescentMode.bBusy) THEN
		fb103StopQuiescentMode(	bStart:= FALSE);
		nStep := 0;
	END_IF
{endregion}
{endregion}

{region "Write"}
1000:	
{region "Enable or Disable Instance"}
	IF (bEnable) THEN
		fb103EnableInstance(bStart := TRUE,
							nAddress := nAddress,
							eAddressType := Tc3_DALI.E_DALIAddressType.Short,
							nInstanceAddress := nInstanceAddress,
							eInstanceAddressType := Tc3_DALI.E_DALIInstanceAddressType.InstanceNumber,
							eCommandPriority := Tc3_DALI.E_DALICommandPriority.Middle);
		IF (NOT fb103EnableInstance.bBusy) THEN
			fb103EnableInstance(bStart := FALSE);
			nStep := 1010;
		END_IF
	ELSE
		fb103DisableInstance(bStart := TRUE,
							 nAddress := nAddress,
							 eAddressType := Tc3_DALI.E_DALIAddressType.Short,
							 nInstanceAddress := nInstanceAddress,
							 eInstanceAddressType := Tc3_DALI.E_DALIInstanceAddressType.InstanceNumber,
							 eCommandPriority := Tc3_DALI.E_DALICommandPriority.Middle);
		IF (NOT fb103DisableInstance.bBusy) THEN
			fb103DisableInstance(bStart := FALSE);
			nStep := 0;
		END_IF
	END_IF
{endregion}
1010:
{region "Set Event Scheme"}
	fb103SetEventScheme(bStart := TRUE,
						nAddress := nAddress,
						eAddressType := Tc3_DALI.E_DALIAddressType.Short,
						nInstanceAddress := nInstanceAddress,
						eInstanceAddressType := Tc3_DALI.E_DALIInstanceAddressType.InstanceNumber,
						eCommandPriority := Tc3_DALI.E_DALICommandPriority.Middle,
						eEventScheme := eEventScheme);
	IF (NOT fb103SetEventScheme.bBusy) THEN
		fb103SetEventScheme(bStart := FALSE);
		nStep := 1020;
	END_IF
{endregion}
1020:
{region "Set Event Filter"}
	nEventFilter.0 := bBit0;
	nEventFilter.1 := bBit1;
	nEventFilter.2 := bBit2;
	nEventFilter.3 := bBit3;
	nEventFilter.4 := bBit4;
	nEventFilter.5 := bBit5;
	nEventFilter.6 := bBit6;
	nEventFilter.7 := bBit7;
	fb103SetEventFilter(bStart := TRUE,
						nAddress := nAddress,
						eAddressType := Tc3_DALI.E_DALIAddressType.Short,
						nInstanceAddress := nInstanceAddress,
						eInstanceAddressType := Tc3_DALI.E_DALIInstanceAddressType.InstanceNumber,
						eCommandPriority := Tc3_DALI.E_DALICommandPriority.Middle,
						nEventFilter := nEventFilter);
	IF (NOT fb103SetEventFilter.bBusy) THEN
		fb103SetEventFilter(bStart := FALSE);
		nStep := 1050;
	END_IF
{endregion}
1050:
{region "Set Event Priority"}
	fb103SetEventPriority(bStart := TRUE,
						  nAddress := nAddress,
						  eAddressType := Tc3_DALI.E_DALIAddressType.Short,
						  nInstanceAddress := nInstanceAddress,
						  eInstanceAddressType := Tc3_DALI.E_DALIInstanceAddressType.InstanceNumber,
						  eCommandPriority := Tc3_DALI.E_DALICommandPriority.Middle,
						  eEventPriority:= eEventPriority);
	IF (NOT fb103SetEventPriority.bBusy) THEN
		fb103SetEventPriority(bStart := FALSE);
		nStep := 0;
	END_IF
{endregion}
{endregion}
2000:
		  fb103IdentifyDevice(bStart := TRUE,
							  nAddress := nAddress,
							  eAddressType := Tc3_DALI.E_DALIAddressType.Short,
		  );
		  IF (NOT fb103IdentifyDevice.bBusy) THEN
				fb103IdentifyDevice(bStart := FALSE);
				  nStep := 0;
		  END_IF
END_CASE
{endregion}
{endregion}

END_FUNCTION_BLOCK

// ---- Tc3_DALI_PLC_Commissioning_Tool/POUs/DALI_PLC_Commissioning/FB_Part301PushButton.TcPOU
FUNCTION_BLOCK FB_Part301PushButton
VAR_INPUT
	ipDALICommunication			:	I_DALICommunication;
END_VAR
VAR_OUTPUT
	bBusy						:	BOOL;
END_VAR
VAR
	{region "Visu"}
	sInputValue					:	STRING[25];
	nInstanceError				:	BYTE;
	nResolution					:	BYTE;
	eEventScheme				:	E_DALIEventScheme;
	nEventFilter				:	DWORD;
	nRepeat						:	UINT(100..2000);
	nStuck						:	BYTE(5..255);
	nShort						:	UINT(0..5100);
	nShortMin					:	UINT;
	nDouble						:	UINT(0..2000);
	nDoubleMin					:	UINT;
	bRead						:	BOOL;
	bWrite						:	BOOL;
	bEnable						:	BOOL;
	bButtonReleased				:	BOOL;
	bButtonPressed				:	BOOL;
	bShortPress					:	BOOL;
	bDoublePress				:	BOOL;
	bLongPressStart				:	BOOL;
	bLongPressRepeat			:	BOOL;
	bLongPressStop				:	BOOL;
	bButtonStuck				:	BOOL;
	bNoRepeatTimer				:	BOOL;
	bNoStuckTimer				:	BOOL;
	bNoShortTimer				:	BOOL;
	bNoDoubleTimer				:	BOOL;
	eEventPriority				:	E_DALIEventPriority := E_DALIEventPriority.Middle;
	{endregion}
	nStep						:	INT;
	nAddress					:	BYTE;
	nInstanceAddress			:	BYTE;
	bHideWaitSymbol				:	BOOL := TRUE;
	nInputValue					:	LWORD;
	nAddressInfo01				:	BYTE;
	nAddressInfo02				:	BYTE;

	fbGetInputNotification		:	FB_DALIGetInputNotification(0);
	fb103StartQuiescentMode		:	FB_DALI103StartQuiescentMode(0);
	fb103StopQuiescentMode		:	FB_DALI103StopQuiescentMode(0);
	fb103QueryInstanceError		:	FB_DALI103QueryInstanceError(0);
	fb103QueryInstanceStatus	:	FB_DALI103QueryInstanceStatus(0);
	fb103QueryResolution		:	FB_DALI103QueryResolution(0);
	fb103QueryInputValue		:	FB_DALI103QueryInputValue(0);
	fb103QueryEventScheme		:	FB_DALI103QueryEventScheme(0);
	fb103QueryEventFilter		:	FB_DALI103QueryEventFilter(0);
	fb103QueryEventPriority		:	FB_DALI103QueryEventPriority(0);
	fb301QueryRepeatTimer		:	FB_DALI301QueryRepeatTimer(0);
	fb301QueryStuckTimer		:	FB_DALI301QueryStuckTimer(0);
	fb301QueryShortTimer		:	FB_DALI301QueryShortTimer(0);
	fb301QueryShortTimerMin		:	FB_DALI301QueryShortTimerMin(0);
	fb301QueryDoubleTimer		:	FB_DALI301QueryDoubleTimer(0);
	fb301QueryDoubleTimerMin	:	FB_DALI301QueryDoubleTimerMin(0);
	fb103EnableInstance			:	FB_DALI103EnableInstance(0);
	fb103DisableInstance		:	FB_DALI103DisableInstance(0);
	fb103SetEventScheme			:	FB_DALI103SetEventScheme(0);
	fb103SetEventFilter			:	FB_DALI103SetEventFilter(0);
	fb103SetEventPriority		:	FB_DALI103SetEventPriority(0);
	fb301SetRepeatTimer			:	FB_DALI301SetRepeatTimer(0);
	fb301SetStuckTimer			:	FB_DALI301SetStuckTimer(0);
	fb301SetShortTimer			:	FB_DALI301SetShortTimer(0);
	fb301SetDoubleTimer			:	FB_DALI301SetDoubleTimer(0);
END_VAR

{region "Detect Commands"}
IF (bRead AND (nStep = 0)) THEN
	nStep := 5;
	bRead := FALSE;
	bHideWaitSymbol := FALSE;
END_IF

IF (bWrite AND (nStep = 0)) THEN
	nStep := 1000;
	bWrite := FALSE;
	bHideWaitSymbol := FALSE;
END_IF
{endregion}
{region "Manage Dialog Selection}
IF (nStep = 0) THEN
	bBusy := FALSE;
ELSE
	bBusy := TRUE;
END_IF
{endregion}
{region "Execute Commands"}
CASE nStep OF
0:
{region "Init"}
	bRead := FALSE;
	bWrite := FALSE;
	bHideWaitSymbol := TRUE;

	fbGetInputNotification.ipDALICommunication := ipDALICommunication;
	fb103StartQuiescentMode.ipDALICommunication := ipDALICommunication;
	fb103StopQuiescentMode.ipDALICommunication := ipDALICommunication;
	fb103QueryInstanceError.ipDALICommunication := ipDALICommunication;
	fb103QueryInstanceStatus.ipDALICommunication := ipDALICommunication;
	fb103QueryResolution.ipDALICommunication := ipDALICommunication;
	fb103QueryInputValue.ipDALICommunication := ipDALICommunication;
	fb103QueryEventScheme.ipDALICommunication := ipDALICommunication;
	fb103QueryEventFilter.ipDALICommunication := ipDALICommunication;
	fb103QueryEventPriority.ipDALICommunication := ipDALICommunication;
	fb301QueryRepeatTimer.ipDALICommunication := ipDALICommunication;
	fb301QueryStuckTimer.ipDALICommunication := ipDALICommunication;
	fb301QueryShortTimer.ipDALICommunication := ipDALICommunication;
	fb301QueryShortTimerMin.ipDALICommunication := ipDALICommunication;
	fb301QueryDoubleTimer.ipDALICommunication := ipDALICommunication;
	fb301QueryDoubleTimerMin.ipDALICommunication := ipDALICommunication;
	fb103EnableInstance.ipDALICommunication := ipDALICommunication;
	fb103DisableInstance.ipDALICommunication := ipDALICommunication;
	fb103SetEventScheme.ipDALICommunication := ipDALICommunication;
	fb103SetEventFilter.ipDALICommunication := ipDALICommunication;
	fb103SetEventPriority.ipDALICommunication := ipDALICommunication;
	fb301SetRepeatTimer.ipDALICommunication := ipDALICommunication;
	fb301SetStuckTimer.ipDALICommunication := ipDALICommunication;
	fb301SetShortTimer.ipDALICommunication := ipDALICommunication;
	fb301SetDoubleTimer.ipDALICommunication := ipDALICommunication;
{endregion}
{region "Read Notifications"}
	CASE eEventScheme OF
	0:
		nAddressInfo01 := 1;
		nAddressInfo02 := nInstanceAddress;
	1:
		nAddressInfo01 := nAddress;
		nAddressInfo02 := 1;
	2:
		nAddressInfo01 := nAddress;
		nAddressInfo02 := nInstanceAddress;
	END_CASE

